	// Process
  E_SEQ_DATABASE.BUCKET_EXIST_CHECK: _m_Seq_BUCKET_EXIST_CHECK();
    IF TRUE
		AND (stSeqCtrlGeneral.eActiveSeqState = E_SEQ_GENERAL.DONE) 
		THEN
			eSeq := E_SEQ_DATABASE.BASE;
		END_IF
  
	E_SEQ_DATABASE.MEASUREMENT_EXIST_CHECK:         _m_Seq_MEASUREMENT_EXIST_CHECK();
    IF TRUE
		AND (stSeqCtrlGeneral.eActiveSeqState = E_SEQ_GENERAL.DONE) 
		THEN
			eSeq := E_SEQ_DATABASE.BASE;
		END_IF
    
  E_SEQ_DATABASE.WRITE_STRUCT:  _m_Seq_WRITE_STRUCT();
    IF TRUE
		AND (stSeqCtrlGeneral.eActiveSeqState = E_SEQ_GENERAL.DONE) 
		THEN
			eSeq := E_SEQ_DATABASE.BASE;
		END_IF
  
  E_SEQ_DATABASE.TAG_EXIST_CHECK:     _m_Seq_TAG_EXIST_CHECK();
    IF TRUE
		AND (stSeqCtrlGeneral.eActiveSeqState = E_SEQ_GENERAL.DONE) 
		THEN
			eSeq := E_SEQ_DATABASE.BASE;
		END_IF
    
  E_SEQ_DATABASE.FIELD_EXIST_CHECK:     _m_Seq_FIELD_EXIST_CHECK();
    IF TRUE
		AND (stSeqCtrlGeneral.eActiveSeqState = E_SEQ_GENERAL.DONE) 
		THEN
			eSeq := E_SEQ_DATABASE.BASE;
		END_IF
    
  E_SEQ_DATABASE.DELETE_MEASUREMENT:    _m_Seq_DELETE_MEASUREMENT();
    IF TRUE
		AND (stSeqCtrlGeneral.eActiveSeqState = E_SEQ_GENERAL.DONE) 
		THEN
			eSeq := E_SEQ_DATABASE.BASE;
		END_IF
    
  E_SEQ_DATABASE.DELETE_ALL_MEASUREMENTS:    _m_Seq_DELETE_ALL_MEASUREMENTS();
    IF TRUE
		AND (stSeqCtrlGeneral.eActiveSeqState = E_SEQ_GENERAL.DONE) 
		THEN
			eSeq := E_SEQ_DATABASE.BASE;
		END_IF
  
  E_SEQ_DATABASE.DELETE_TAG:    _m_Seq_DELETE_TAG();
    IF TRUE
		AND (stSeqCtrlGeneral.eActiveSeqState = E_SEQ_GENERAL.DONE) 
		THEN
			eSeq := E_SEQ_DATABASE.BASE;
		END_IF
    
  E_SEQ_DATABASE.DELETE_TAG_CONTENT_BLOCK:    _m_Seq_DELETE_TAG_CONTENT_BLOCK();
    IF TRUE
		AND (stSeqCtrlGeneral.eActiveSeqState = E_SEQ_GENERAL.DONE) 
		THEN
			eSeq := E_SEQ_DATABASE.BASE;
		END_IF
  
  E_SEQ_DATABASE.DELETE_FIELD:           _m_Seq_DELETE_FIELD();
    IF TRUE
		AND (stSeqCtrlGeneral.eActiveSeqState = E_SEQ_GENERAL.DONE) 
		THEN
			eSeq := E_SEQ_DATABASE.BASE;
		END_IF
    
  E_SEQ_DATABASE.GET_TOTAL_MEASUREMENTS:           _m_Seq_GET_TOTAL_MEASUREMENTS();
    IF TRUE
		AND (stSeqCtrlGeneral.eActiveSeqState = E_SEQ_GENERAL.DONE) 
		THEN
			eSeq := E_SEQ_DATABASE.BASE;
		END_IF

  // End
	E_SEQ_DATABASE.END:;
	E_SEQ_DATABASE.ERROR_SEQ:;	
END_CASE

strTemp:=TO_STRING(eSeq);

METHOD PRIVATE _m_DebugManager
VAR_INPUT
	iStepID: int;
END_VAR
IF TRUE
AND THIS^.stSeqCtrlGeneral.bDebugModeActive 
AND NOT THIS^.stSeqCtrlGeneral.bActiveStep
THEN


THIS^.stSeqCtrlGeneral.bBreakpointActive:=FALSE;

FOR i:=0 TO 10 DO
	
	IF TRUE
	AND iStepID=THIS^.stSeqCtrlGeneral.listBreakpoint[i] 
	AND iStepID<>0
	THEN
		EXIT;
	END_IF
END_FOR
IF (i<=10) THEN
	THIS^.stSeqCtrlGeneral.bBreakpointActive:=TRUE;
END_IF

END_IF
END_METHOD

METHOD PRIVATE _m_Delay : BOOL
VAR_INPUT
	DelayTime:	TIME;
END_VAR
THIS^.stSeqCtrlGeneral.bDelayActive:=TRUE;
THIS^.stSeqCtrlGeneral.tDelay:=DelayTime;
_m_Delay:=FALSE;
IF THIS^.stSeqCtrlGeneral.tonDelay.Q THEN
	_m_Delay:=TRUE;
END_IF
END_METHOD

METHOD PRIVATE _m_GeneralStepSetting : BOOL
VAR_INPUT
	StepType:			    	E_STEP_STATE_TYPE;
	InfoTextID:					STRING(20);
	EnableDebug:	   			BOOL;	
	
END_VAR
IF THIS^.stSeqCtrlGeneral.bActiveStep THEN
	THIS^.stSeqCtrlGeneral.eStep_Type:=StepType;
	THIS^.stSeqCtrlGeneral.strExtraInfo:= GenLib.F_RET_TXTLIST_ENTRY(strPortNr:='851',strID:='',strTxtLstName:=InfoTextID);
END_IF
END_METHOD

METHOD PRIVATE _m_SaveLastStep : BOOL
VAR_INPUT
END_VAR
VAR
	i: dint;
END_VAR
IF NOT THIS^.stSeqCtrlGeneral.bActiveStep THEN
	
	FOR i:=49 TO 1 BY -1 DO
			stSeqCtrlGeneral.listLastSteps[i].strStepName:=stSeqCtrlGeneral.listLastSteps[i-1].strStepName;
			stSeqCtrlGeneral.listLastSteps[i].tStepTime:=stSeqCtrlGeneral.listLastSteps[i-1].tStepTime;
			stSeqCtrlGeneral.listLastSteps[i].tDelayTime:=stSeqCtrlGeneral.listLastSteps[i-1].tDelayTime;
	END_FOR
	stSeqCtrlGeneral.listLastSteps[0].strStepName:=TO_STRING(THIS^.eSeq);
	stSeqCtrlGeneral.listLastSteps[1].tStepTime:=THIS^.stSeqCtrlGeneral.tonStepTime.ET;
	stSeqCtrlGeneral.listLastSteps[1].tStepTime:=THIS^.stSeqCtrlGeneral.tonDelay.ET;
ELSE
	stSeqCtrlGeneral.listLastSteps[0].tStepTime:=THIS^.stSeqCtrlGeneral.tonStepTime.ET;
	stSeqCtrlGeneral.listLastSteps[0].tDelayTime:=THIS^.stSeqCtrlGeneral.tonDelay.ET;	
END_IF
END_METHOD

METHOD PRIVATE _m_Seq_BUCKET_EXIST_CHECK : E_SEQ_PROCESS
VAR_INPUT
END_VAR
VAR
	ActiveSeq: STRING;
END_VAR
//THIS^._m_GeneralStepSetting(StepType:=E_STEP_STATE_TYPE.INIT,
ActiveSeq := TO_STRING(THIS^.eSeq);

CASE THIS^.stSeqCtrlGeneral.eActiveSeqState OF
E_SEQ_GENERAL.READY:;
	
E_SEQ_GENERAL.EXECUTE:;
	IF TRUE
	THEN
		THIS^.stSeqCtrlGeneral.eActiveSeqState := E_SEQ_GENERAL.RESET;
	END_IF
  
E_SEQ_GENERAL.RESET:;
	THIS^.stSeqCtrlGeneral.iInternalSeqStateCase := 0;
	IF TRUE
	THEN
    THIS^.bResult := FALSE;
		THIS^.stSeqCtrlGeneral.eActiveSeqState := E_SEQ_GENERAL.BUSY;
	END_IF
  
E_SEQ_GENERAL.BUSY:;
	CASE THIS^.stSeqCtrlGeneral.iInternalSeqStateCase OF
    0:  // Execute
      IF TRUE 
      AND THIS^.bAdsConnected
      AND NOT THIS^.bBusy
      AND THIS^.bReady
			THEN 
        THIS^.bGetBucketExist := TRUE;
        THIS^.stSeqCtrlGeneral.iInternalSeqStateCase := 10;
			END_IF

    10:	// Wait for done
      IF TRUE 
      AND NOT THIS^.bBusy
      AND THIS^.bReady
      AND NOT THIS^.bGetBucketExist
			THEN 
        THIS^.stSeqCtrlGeneral.iInternalSeqStateCase := 1000;
			END_IF
      
    1000: // Exit step
      IF TRUE
      THEN
        THIS^.stSeqCtrlGeneral.iInternalSeqStateCase := 9999;
			END_IF
      
	ELSE
		THIS^.stSeqCtrlGeneral.eActiveSeqState := E_SEQ_GENERAL.DONE;  
	END_CASE
	THIS^.stSeqCtrlGeneral.strExtraInfo := CONCAT('Internal state: ', TO_STRING(THIS^.stSeqCtrlGeneral.iInternalSeqStateCase));

E_SEQ_GENERAL.DONE:;

E_SEQ_GENERAL.ERROR:;

E_SEQ_GENERAL.TIME_OUT:; 

ELSE
  THIS^.stSeqCtrlGeneral.eActiveSeqState := E_SEQ_GENERAL.ERROR;
END_CASE
END_METHOD

METHOD PRIVATE _m_Seq_CLEAR_MEASUREMENT : E_SEQ_PROCESS
VAR_INPUT
END_VAR
VAR
	ActiveSeq: STRING;
END_VAR
//THIS^._m_GeneralStepSetting(StepType:=E_STEP_STATE_TYPE.INIT,
ActiveSeq := TO_STRING(THIS^.eSeq);

CASE THIS^.stSeqCtrlGeneral.eActiveSeqState OF
E_SEQ_GENERAL.READY:;
	
E_SEQ_GENERAL.EXECUTE:;
	IF TRUE
	THEN
		THIS^.stSeqCtrlGeneral.eActiveSeqState := E_SEQ_GENERAL.RESET;
	END_IF
  
E_SEQ_GENERAL.RESET:;
	THIS^.stSeqCtrlGeneral.iInternalSeqStateCase := 0;
	IF TRUE
	THEN
    THIS^.bResult := FALSE;
		THIS^.stSeqCtrlGeneral.eActiveSeqState := E_SEQ_GENERAL.BUSY;
	END_IF
  
E_SEQ_GENERAL.BUSY:;
	CASE THIS^.stSeqCtrlGeneral.iInternalSeqStateCase OF
		0:	// Entrance step --> Create command
      IF TRUE 
      AND THIS^.bAdsConnected
      AND NOT THIS^.bBusy
      AND THIS^.bReady
			THEN 
        THIS^.bClearMeasurement := TRUE;
        THIS^.stSeqCtrlGeneral.iInternalSeqStateCase := 10;
			END_IF
      
    10:	// Wait for done
      IF TRUE 
      AND NOT THIS^.bBusy
      AND THIS^.bReady
      AND NOT THIS^.bClearMeasurement
			THEN 
        THIS^.stSeqCtrlGeneral.iInternalSeqStateCase := 1000;
			END_IF
      
    1000: // Exit step
      IF TRUE
      THEN
        THIS^.stSeqCtrlGeneral.iInternalSeqStateCase := 9999;
			END_IF
      
	ELSE
		THIS^.stSeqCtrlGeneral.eActiveSeqState := E_SEQ_GENERAL.DONE;  
	END_CASE
	THIS^.stSeqCtrlGeneral.strExtraInfo := CONCAT('Internal state: ', TO_STRING(THIS^.stSeqCtrlGeneral.iInternalSeqStateCase));

E_SEQ_GENERAL.DONE:;

E_SEQ_GENERAL.ERROR:;

E_SEQ_GENERAL.TIME_OUT:; 
IF TRUE
AND THIS^.stSeqCtrlGeneral.bTimeOutActiveQuit 
THEN
  THIS^.stSeqCtrlGeneral.strExtraInfo := 'Bitte quittieren und erneut testen';
  IF TRUE
  //AND itfOpMode.P_QUIT
  THEN
    THIS^.stSeqCtrlGeneral.eActiveSeqState := E_SEQ_GENERAL.EXECUTE;
	END_IF
  
END_IF

ELSE
  THIS^.stSeqCtrlGeneral.eActiveSeqState := E_SEQ_GENERAL.ERROR;
END_CASE
END_METHOD

METHOD PRIVATE _m_Seq_DELETE_ALL_MEASUREMENTS : E_SEQ_PROCESS
VAR_INPUT
END_VAR
VAR
	ActiveSeq: STRING;
END_VAR
//THIS^._m_GeneralStepSetting(StepType:=E_STEP_STATE_TYPE.INIT,
ActiveSeq := TO_STRING(THIS^.eSeq);

CASE THIS^.stSeqCtrlGeneral.eActiveSeqState OF
E_SEQ_GENERAL.READY:;

E_SEQ_GENERAL.EXECUTE:;
	IF TRUE
	THEN
		THIS^.stSeqCtrlGeneral.eActiveSeqState := E_SEQ_GENERAL.RESET;
	END_IF
  
E_SEQ_GENERAL.RESET:;
	THIS^.stSeqCtrlGeneral.iInternalSeqStateCase := 0;
	IF TRUE
	THEN
    THIS^.bResult := FALSE;
		THIS^.stSeqCtrlGeneral.eActiveSeqState := E_SEQ_GENERAL.BUSY;
	END_IF
  
E_SEQ_GENERAL.BUSY:;
	CASE THIS^.stSeqCtrlGeneral.iInternalSeqStateCase OF
		0:	// Entrance step --> Create command
      IF TRUE 
      AND THIS^.bAdsConnected
      AND NOT THIS^.bBusy
      AND THIS^.bReady
			THEN 
        THIS^.bDeleteAllMeasurements := TRUE;
        THIS^.stSeqCtrlGeneral.iInternalSeqStateCase := 10;
			END_IF
      
    10:	// Wait for done
      IF TRUE 
      AND NOT THIS^.bBusy
      AND THIS^.bReady
      AND NOT THIS^.bDeleteAllMeasurements
			THEN 
        THIS^.stSeqCtrlGeneral.iInternalSeqStateCase := 1000;
			END_IF
      
    1000: // Exit step
      IF TRUE
      THEN
        THIS^.stSeqCtrlGeneral.iInternalSeqStateCase := 9999;
			END_IF
      
	ELSE
		THIS^.stSeqCtrlGeneral.eActiveSeqState := E_SEQ_GENERAL.DONE;  
	END_CASE
	THIS^.stSeqCtrlGeneral.strExtraInfo := CONCAT('Internal state: ', TO_STRING(THIS^.stSeqCtrlGeneral.iInternalSeqStateCase));

E_SEQ_GENERAL.DONE:;

E_SEQ_GENERAL.ERROR:;

E_SEQ_GENERAL.TIME_OUT:; 
IF TRUE
AND THIS^.stSeqCtrlGeneral.bTimeOutActiveQuit 
THEN
  THIS^.stSeqCtrlGeneral.strExtraInfo := 'Bitte quittieren und erneut testen';
  IF TRUE
  //AND itfOpMode.P_QUIT
  THEN
    THIS^.stSeqCtrlGeneral.eActiveSeqState := E_SEQ_GENERAL.EXECUTE;
	END_IF
  
END_IF

ELSE
  THIS^.stSeqCtrlGeneral.eActiveSeqState := E_SEQ_GENERAL.ERROR;
END_CASE
END_METHOD

METHOD PRIVATE _m_Seq_DELETE_FIELD : E_SEQ_PROCESS
VAR_INPUT
END_VAR
VAR
	ActiveSeq: STRING;
END_VAR
//THIS^._m_GeneralStepSetting(StepType:=E_STEP_STATE_TYPE.INIT,
ActiveSeq := TO_STRING(THIS^.eSeq);

CASE THIS^.stSeqCtrlGeneral.eActiveSeqState OF
E_SEQ_GENERAL.READY:;
	
E_SEQ_GENERAL.EXECUTE:;
	IF TRUE
	THEN
		THIS^.stSeqCtrlGeneral.eActiveSeqState := E_SEQ_GENERAL.RESET;
	END_IF
  
E_SEQ_GENERAL.RESET:;
	THIS^.stSeqCtrlGeneral.iInternalSeqStateCase := 0;
	IF TRUE
	THEN
    THIS^.bResult := FALSE;
		THIS^.stSeqCtrlGeneral.eActiveSeqState := E_SEQ_GENERAL.BUSY;
	END_IF
  
E_SEQ_GENERAL.BUSY:;
	CASE THIS^.stSeqCtrlGeneral.iInternalSeqStateCase OF
    0:  // Execute
      IF TRUE 
      AND THIS^.bAdsConnected
      AND NOT THIS^.bBusy
      AND THIS^.bReady
			THEN 
        THIS^.bDeleteField := TRUE;
        THIS^.stSeqCtrlGeneral.iInternalSeqStateCase := 10;
			END_IF

    10:	// Wait for done
      IF TRUE 
      AND NOT THIS^.bBusy
      AND THIS^.bReady
      AND NOT THIS^.bDeleteField
			THEN 
        THIS^.stSeqCtrlGeneral.iInternalSeqStateCase := 1000;
			END_IF
      
    1000: // Exit step
      IF TRUE
      THEN
        THIS^.stSeqCtrlGeneral.iInternalSeqStateCase := 9999;
			END_IF
      
	ELSE
		THIS^.stSeqCtrlGeneral.eActiveSeqState := E_SEQ_GENERAL.DONE;  
	END_CASE
	THIS^.stSeqCtrlGeneral.strExtraInfo := CONCAT('Internal state: ', TO_STRING(THIS^.stSeqCtrlGeneral.iInternalSeqStateCase));

E_SEQ_GENERAL.DONE:;

E_SEQ_GENERAL.ERROR:;

E_SEQ_GENERAL.TIME_OUT:; 

ELSE
  THIS^.stSeqCtrlGeneral.eActiveSeqState := E_SEQ_GENERAL.ERROR;
END_CASE
END_METHOD

METHOD PRIVATE _m_Seq_DELETE_MEASUREMENT : E_SEQ_PROCESS
VAR_INPUT
END_VAR
VAR
	ActiveSeq: STRING;
END_VAR
//THIS^._m_GeneralStepSetting(StepType:=E_STEP_STATE_TYPE.INIT,
ActiveSeq := TO_STRING(THIS^.eSeq);

CASE THIS^.stSeqCtrlGeneral.eActiveSeqState OF
E_SEQ_GENERAL.READY:;
	
E_SEQ_GENERAL.EXECUTE:;
	IF TRUE
	THEN
		THIS^.stSeqCtrlGeneral.eActiveSeqState := E_SEQ_GENERAL.RESET;
	END_IF
  
E_SEQ_GENERAL.RESET:;
	THIS^.stSeqCtrlGeneral.iInternalSeqStateCase := 0;
	IF TRUE
	THEN
    THIS^.bResult := FALSE;
		THIS^.stSeqCtrlGeneral.eActiveSeqState := E_SEQ_GENERAL.BUSY;
	END_IF
  
E_SEQ_GENERAL.BUSY:;
	CASE THIS^.stSeqCtrlGeneral.iInternalSeqStateCase OF
		0:	// Entrance step --> Create command
      IF TRUE 
      AND THIS^.bAdsConnected
      AND NOT THIS^.bBusy
      AND THIS^.bReady
			THEN 
        THIS^.bDeleteMeasurement := TRUE;
        THIS^.stSeqCtrlGeneral.iInternalSeqStateCase := 10;
			END_IF
      
    10:	// Wait for done
      IF TRUE 
      AND NOT THIS^.bBusy
      AND THIS^.bReady
      AND NOT THIS^.bDeleteMeasurement
			THEN 
        THIS^.stSeqCtrlGeneral.iInternalSeqStateCase := 1000;
			END_IF
      
    1000: // Exit step
      IF TRUE
      THEN
        THIS^.stSeqCtrlGeneral.iInternalSeqStateCase := 9999;
			END_IF
      
	ELSE
		THIS^.stSeqCtrlGeneral.eActiveSeqState := E_SEQ_GENERAL.DONE;  
	END_CASE
	THIS^.stSeqCtrlGeneral.strExtraInfo := CONCAT('Internal state: ', TO_STRING(THIS^.stSeqCtrlGeneral.iInternalSeqStateCase));

E_SEQ_GENERAL.DONE:;

E_SEQ_GENERAL.ERROR:;

E_SEQ_GENERAL.TIME_OUT:; 
IF TRUE
AND THIS^.stSeqCtrlGeneral.bTimeOutActiveQuit 
THEN
  THIS^.stSeqCtrlGeneral.strExtraInfo := 'Bitte quittieren und erneut testen';
  IF TRUE
  //AND itfOpMode.P_QUIT
  THEN
    THIS^.stSeqCtrlGeneral.eActiveSeqState := E_SEQ_GENERAL.EXECUTE;
	END_IF
  
END_IF

ELSE
  THIS^.stSeqCtrlGeneral.eActiveSeqState := E_SEQ_GENERAL.ERROR;
END_CASE
END_METHOD

METHOD PRIVATE _m_Seq_DELETE_TAG : E_SEQ_PROCESS
VAR_INPUT
END_VAR
VAR
	ActiveSeq: STRING;
END_VAR
//THIS^._m_GeneralStepSetting(StepType:=E_STEP_STATE_TYPE.INIT,
ActiveSeq := TO_STRING(THIS^.eSeq);

CASE THIS^.stSeqCtrlGeneral.eActiveSeqState OF
E_SEQ_GENERAL.READY:;
	
E_SEQ_GENERAL.EXECUTE:;
	IF TRUE
	THEN
		THIS^.stSeqCtrlGeneral.eActiveSeqState := E_SEQ_GENERAL.RESET;
	END_IF
  
E_SEQ_GENERAL.RESET:;
	THIS^.stSeqCtrlGeneral.iInternalSeqStateCase := 0;
	IF TRUE
	THEN
    THIS^.bResult := FALSE;
		THIS^.stSeqCtrlGeneral.eActiveSeqState := E_SEQ_GENERAL.BUSY;
	END_IF
  
E_SEQ_GENERAL.BUSY:;
	CASE THIS^.stSeqCtrlGeneral.iInternalSeqStateCase OF
    0:  // Execute
      IF TRUE 
      AND THIS^.bAdsConnected
      AND NOT THIS^.bBusy
      AND THIS^.bReady
			THEN 
        THIS^.bDeleteTag := TRUE;
        THIS^.stSeqCtrlGeneral.iInternalSeqStateCase := 10;
			END_IF

    10:	// Wait for done
      IF TRUE 
      AND NOT THIS^.bBusy
      AND THIS^.bReady
      AND NOT THIS^.bDeleteTag
			THEN 
        THIS^.stSeqCtrlGeneral.iInternalSeqStateCase := 1000;
			END_IF
      
    1000: // Exit step
      IF TRUE
      THEN
        THIS^.stSeqCtrlGeneral.iInternalSeqStateCase := 9999;
			END_IF
      
	ELSE
		THIS^.stSeqCtrlGeneral.eActiveSeqState := E_SEQ_GENERAL.DONE;  
	END_CASE
	THIS^.stSeqCtrlGeneral.strExtraInfo := CONCAT('Internal state: ', TO_STRING(THIS^.stSeqCtrlGeneral.iInternalSeqStateCase));

E_SEQ_GENERAL.DONE:;

E_SEQ_GENERAL.ERROR:;

E_SEQ_GENERAL.TIME_OUT:; 

ELSE
  THIS^.stSeqCtrlGeneral.eActiveSeqState := E_SEQ_GENERAL.ERROR;
END_CASE
END_METHOD

METHOD PRIVATE _m_Seq_DELETE_TAG_CONTENT_BLOCK : E_SEQ_PROCESS
VAR_INPUT
END_VAR
VAR
	ActiveSeq: STRING;
END_VAR
//THIS^._m_GeneralStepSetting(StepType:=E_STEP_STATE_TYPE.INIT,
ActiveSeq := TO_STRING(THIS^.eSeq);

CASE THIS^.stSeqCtrlGeneral.eActiveSeqState OF
E_SEQ_GENERAL.READY:;
	
E_SEQ_GENERAL.EXECUTE:;
	IF TRUE
	THEN
		THIS^.stSeqCtrlGeneral.eActiveSeqState := E_SEQ_GENERAL.RESET;
	END_IF
  
E_SEQ_GENERAL.RESET:;
	THIS^.stSeqCtrlGeneral.iInternalSeqStateCase := 0;
	IF TRUE
	THEN
    THIS^.bResult := FALSE;
		THIS^.stSeqCtrlGeneral.eActiveSeqState := E_SEQ_GENERAL.BUSY;
	END_IF
  
E_SEQ_GENERAL.BUSY:;
	CASE THIS^.stSeqCtrlGeneral.iInternalSeqStateCase OF
    0:  // Execute
      IF TRUE 
      AND THIS^.bAdsConnected
      AND NOT THIS^.bBusy
      AND THIS^.bReady
			THEN 
        THIS^.bDeleteTagContentBlock := TRUE;
        THIS^.stSeqCtrlGeneral.iInternalSeqStateCase := 10;
			END_IF

    10:	// Wait for done
      IF TRUE 
      AND NOT THIS^.bBusy
      AND THIS^.bReady
      AND NOT THIS^.bDeleteTagContentBlock
			THEN 
        THIS^.stSeqCtrlGeneral.iInternalSeqStateCase := 1000;
			END_IF
      
    1000: // Exit step
      IF TRUE
      THEN
        THIS^.stSeqCtrlGeneral.iInternalSeqStateCase := 9999;
			END_IF
      
	ELSE
		THIS^.stSeqCtrlGeneral.eActiveSeqState := E_SEQ_GENERAL.DONE;  
	END_CASE
	THIS^.stSeqCtrlGeneral.strExtraInfo := CONCAT('Internal state: ', TO_STRING(THIS^.stSeqCtrlGeneral.iInternalSeqStateCase));

E_SEQ_GENERAL.DONE:;

E_SEQ_GENERAL.ERROR:;

E_SEQ_GENERAL.TIME_OUT:; 

ELSE
  THIS^.stSeqCtrlGeneral.eActiveSeqState := E_SEQ_GENERAL.ERROR;
END_CASE
END_METHOD

METHOD PRIVATE _m_Seq_FIELD_EXIST_CHECK : E_SEQ_PROCESS
VAR_INPUT
END_VAR
VAR
	ActiveSeq: STRING;
END_VAR
//THIS^._m_GeneralStepSetting(StepType:=E_STEP_STATE_TYPE.INIT,
ActiveSeq := TO_STRING(THIS^.eSeq);

CASE THIS^.stSeqCtrlGeneral.eActiveSeqState OF
E_SEQ_GENERAL.READY:;
	
E_SEQ_GENERAL.EXECUTE:;
	IF TRUE
	THEN
		THIS^.stSeqCtrlGeneral.eActiveSeqState := E_SEQ_GENERAL.RESET;
	END_IF
  
E_SEQ_GENERAL.RESET:;
	THIS^.stSeqCtrlGeneral.iInternalSeqStateCase := 0;
	IF TRUE
	THEN
    THIS^.bResult := FALSE;
		THIS^.stSeqCtrlGeneral.eActiveSeqState := E_SEQ_GENERAL.BUSY;
	END_IF
  
E_SEQ_GENERAL.BUSY:;
	CASE THIS^.stSeqCtrlGeneral.iInternalSeqStateCase OF
    0:  // Execute
      IF TRUE 
      AND THIS^.bAdsConnected
      AND NOT THIS^.bBusy
      AND THIS^.bReady
			THEN 
        THIS^.bGetFieldExist := TRUE;
        THIS^.stSeqCtrlGeneral.iInternalSeqStateCase := 10;
			END_IF

    10:	// Wait for done
      IF TRUE 
      AND NOT THIS^.bBusy
      AND THIS^.bReady
      AND NOT THIS^.bGetFieldExist
			THEN 
        THIS^.stSeqCtrlGeneral.iInternalSeqStateCase := 1000;
			END_IF
      
    1000: // Exit step
      IF TRUE
      THEN
        THIS^.stSeqCtrlGeneral.iInternalSeqStateCase := 9999;
			END_IF
      
	ELSE
		THIS^.stSeqCtrlGeneral.eActiveSeqState := E_SEQ_GENERAL.DONE;  
	END_CASE
	THIS^.stSeqCtrlGeneral.strExtraInfo := CONCAT('Internal state: ', TO_STRING(THIS^.stSeqCtrlGeneral.iInternalSeqStateCase));

E_SEQ_GENERAL.DONE:;

E_SEQ_GENERAL.ERROR:;

E_SEQ_GENERAL.TIME_OUT:; 

ELSE
  THIS^.stSeqCtrlGeneral.eActiveSeqState := E_SEQ_GENERAL.ERROR;
END_CASE
END_METHOD

METHOD PRIVATE _m_Seq_GET_TOTAL_MEASUREMENTS : E_SEQ_PROCESS
VAR_INPUT
END_VAR
VAR
	ActiveSeq: STRING;
END_VAR
//THIS^._m_GeneralStepSetting(StepType:=E_STEP_STATE_TYPE.INIT,
ActiveSeq := TO_STRING(THIS^.eSeq);

CASE THIS^.stSeqCtrlGeneral.eActiveSeqState OF
E_SEQ_GENERAL.READY:;
	
E_SEQ_GENERAL.EXECUTE:;
	IF TRUE
	THEN
		THIS^.stSeqCtrlGeneral.eActiveSeqState := E_SEQ_GENERAL.RESET;
	END_IF
  
E_SEQ_GENERAL.RESET:;
	THIS^.stSeqCtrlGeneral.iInternalSeqStateCase := 0;
	IF TRUE
	THEN
    THIS^.bResult := FALSE;
		THIS^.stSeqCtrlGeneral.eActiveSeqState := E_SEQ_GENERAL.BUSY;
	END_IF
  
E_SEQ_GENERAL.BUSY:;
	CASE THIS^.stSeqCtrlGeneral.iInternalSeqStateCase OF
    0:  // Execute
      IF TRUE 
      AND THIS^.bAdsConnected
      AND NOT THIS^.bBusy
      AND THIS^.bReady
			THEN 
        THIS^.bGetTotalMeasurements := TRUE;
        THIS^.stSeqCtrlGeneral.iInternalSeqStateCase := 10;
			END_IF

    10:	// Wait for done
      IF TRUE 
      AND NOT THIS^.bBusy
      AND THIS^.bReady
      AND NOT THIS^.bGetTotalMeasurements
			THEN 
        THIS^.stSeqCtrlGeneral.iInternalSeqStateCase := 1000;
			END_IF
      
    1000: // Exit step
      IF TRUE
      THEN
        THIS^.stSeqCtrlGeneral.iInternalSeqStateCase := 9999;
			END_IF
      
	ELSE
		THIS^.stSeqCtrlGeneral.eActiveSeqState := E_SEQ_GENERAL.DONE;  
	END_CASE
	THIS^.stSeqCtrlGeneral.strExtraInfo := CONCAT('Internal state: ', TO_STRING(THIS^.stSeqCtrlGeneral.iInternalSeqStateCase));

E_SEQ_GENERAL.DONE:;

E_SEQ_GENERAL.ERROR:;

E_SEQ_GENERAL.TIME_OUT:; 

ELSE
  THIS^.stSeqCtrlGeneral.eActiveSeqState := E_SEQ_GENERAL.ERROR;
END_CASE
END_METHOD

METHOD PRIVATE _m_Seq_INIT : E_SEQ_PROCESS
VAR_INPUT
END_VAR
VAR
	ActiveSeq: STRING;
END_VAR
VAR
	
END_VAR
//THIS^._m_GeneralStepSetting(StepType:=E_STEP_STATE_TYPE.INIT,
ActiveSeq := TO_STRING(THIS^.eSeq);

CASE THIS^.stSeqCtrlGeneral.eActiveSeqState OF
E_SEQ_GENERAL.READY:;
	
E_SEQ_GENERAL.EXECUTE:;
	IF TRUE
	THEN
		THIS^.stSeqCtrlGeneral.eActiveSeqState := E_SEQ_GENERAL.RESET;
	END_IF
E_SEQ_GENERAL.RESET:;
	THIS^.stSeqCtrlGeneral.iInternalSeqStateCase := 0;
	IF TRUE
	THEN
		THIS^.stSeqCtrlGeneral.eActiveSeqState := E_SEQ_GENERAL.BUSY;
	END_IF
E_SEQ_GENERAL.BUSY:;
	CASE THIS^.stSeqCtrlGeneral.iInternalSeqStateCase OF
		0:	// Entrance step
      IF TRUE
			THEN 
        THIS^.bResult := FALSE;
        THIS^.bGetBucketExist := FALSE;
        THIS^.sBucketName := '';
        THIS^.bGetMeasurementExist := FALSE;
        THIS^.sMeasurementName := '';
        THIS^.bDeleteMeasurement := FALSE;
        THIS^.bDeleteAllMeasurements := FALSE;
        THIS^.bWriteStructData := FALSE;
        THIS^.sTagName := '';
        THIS^.sFieldName := '';
        //THIS^.stFieldValues := '';
        //FOR THIS^.i := 0 TO TO_INT(SIZEOF(arrFieldNames)) BY 1 DO
        //  THIS^.arrFieldNames[i] := '';
        //  THIS^.arrFieldStructContent[i] := '';
        //END_FOR
        THIS^.dtFrom := DT#1970-1-1-0:0:0;
        THIS^.dtTo := DT#1970-1-1-0:0:0;
				THIS^.stSeqCtrlGeneral.iInternalSeqStateCase := 1000;
			END_IF
      
    1000:	// Exit step
      IF TRUE
			THEN
        THIS^.stSeqCtrlGeneral.iInternalSeqStateCase := 9999;
      END_IF
      
	ELSE
		THIS^.stSeqCtrlGeneral.eActiveSeqState := E_SEQ_GENERAL.DONE;  
	END_CASE
	THIS^.stSeqCtrlGeneral.strExtraInfo := CONCAT('Internal state: ', TO_STRING(THIS^.stSeqCtrlGeneral.iInternalSeqStateCase));
E_SEQ_GENERAL.DONE:;
E_SEQ_GENERAL.ERROR:;
E_SEQ_GENERAL.TIME_OUT:; 

IF TRUE
AND THIS^.stSeqCtrlGeneral.bTimeOutActiveQuit 
THEN
  THIS^.stSeqCtrlGeneral.strExtraInfo := 'Bitte quittieren und erneut testen';
  IF TRUE
  //AND itfOpMode.P_QUIT
  THEN
    THIS^.stSeqCtrlGeneral.eActiveSeqState := E_SEQ_GENERAL.EXECUTE;
	END_IF
  
END_IF

ELSE
  THIS^.stSeqCtrlGeneral.eActiveSeqState := E_SEQ_GENERAL.ERROR;
END_CASE
END_METHOD

METHOD PRIVATE _m_Seq_MEASUREMENT_EXIST_CHECK : E_SEQ_PROCESS
VAR_INPUT
END_VAR
VAR
	ActiveSeq: STRING;
END_VAR
//THIS^._m_GeneralStepSetting(StepType:=E_STEP_STATE_TYPE.INIT,
ActiveSeq := TO_STRING(THIS^.eSeq);

CASE THIS^.stSeqCtrlGeneral.eActiveSeqState OF
E_SEQ_GENERAL.READY:;
	
E_SEQ_GENERAL.EXECUTE:;
	IF TRUE
	THEN
		THIS^.stSeqCtrlGeneral.eActiveSeqState := E_SEQ_GENERAL.RESET;
	END_IF
  
E_SEQ_GENERAL.RESET:;
	THIS^.stSeqCtrlGeneral.iInternalSeqStateCase := 0;
	IF TRUE
	THEN
    THIS^.bResult := FALSE;
		THIS^.stSeqCtrlGeneral.eActiveSeqState := E_SEQ_GENERAL.BUSY;
	END_IF
  
E_SEQ_GENERAL.BUSY:;
	CASE THIS^.stSeqCtrlGeneral.iInternalSeqStateCase OF
    0:  // Execute
      IF TRUE 
      AND THIS^.bAdsConnected
      AND NOT THIS^.bBusy
      AND THIS^.bReady
			THEN 
        THIS^.bGetMeasurementExist := TRUE;
        THIS^.stSeqCtrlGeneral.iInternalSeqStateCase := 10;
			END_IF

    10:	// Wait for done
      IF TRUE 
      AND NOT THIS^.bBusy
      AND THIS^.bReady
      AND NOT THIS^.bGetMeasurementExist
			THEN 
        THIS^.stSeqCtrlGeneral.iInternalSeqStateCase := 1000;
			END_IF
      
    1000: // Exit step
      IF TRUE
      THEN
        THIS^.stSeqCtrlGeneral.iInternalSeqStateCase := 9999;
			END_IF
      
	ELSE
		THIS^.stSeqCtrlGeneral.eActiveSeqState := E_SEQ_GENERAL.DONE;  
	END_CASE
	THIS^.stSeqCtrlGeneral.strExtraInfo := CONCAT('Internal state: ', TO_STRING(THIS^.stSeqCtrlGeneral.iInternalSeqStateCase));

E_SEQ_GENERAL.DONE:;

E_SEQ_GENERAL.ERROR:;

E_SEQ_GENERAL.TIME_OUT:; 

ELSE
  THIS^.stSeqCtrlGeneral.eActiveSeqState := E_SEQ_GENERAL.ERROR;
END_CASE
END_METHOD

METHOD PRIVATE _m_Seq_TAG_EXIST_CHECK : E_SEQ_PROCESS
VAR_INPUT
END_VAR
VAR
	ActiveSeq: STRING;
END_VAR
//THIS^._m_GeneralStepSetting(StepType:=E_STEP_STATE_TYPE.INIT,
ActiveSeq := TO_STRING(THIS^.eSeq);

CASE THIS^.stSeqCtrlGeneral.eActiveSeqState OF
E_SEQ_GENERAL.READY:;
	
E_SEQ_GENERAL.EXECUTE:;
	IF TRUE
	THEN
		THIS^.stSeqCtrlGeneral.eActiveSeqState := E_SEQ_GENERAL.RESET;
	END_IF
  
E_SEQ_GENERAL.RESET:;
	THIS^.stSeqCtrlGeneral.iInternalSeqStateCase := 0;
	IF TRUE
	THEN
    THIS^.bResult := FALSE;
		THIS^.stSeqCtrlGeneral.eActiveSeqState := E_SEQ_GENERAL.BUSY;
	END_IF
  
E_SEQ_GENERAL.BUSY:;
	CASE THIS^.stSeqCtrlGeneral.iInternalSeqStateCase OF
    0:  // Execute
      IF TRUE 
      AND THIS^.bAdsConnected
      AND NOT THIS^.bBusy
      AND THIS^.bReady
			THEN 
        THIS^.bGetTagExist := TRUE;
        THIS^.stSeqCtrlGeneral.iInternalSeqStateCase := 10;
			END_IF

    10:	// Wait for done
      IF TRUE 
      AND NOT THIS^.bBusy
      AND THIS^.bReady
      AND NOT THIS^.bGetTagExist
			THEN 
        THIS^.stSeqCtrlGeneral.iInternalSeqStateCase := 1000;
			END_IF
      
    1000: // Exit step
      IF TRUE
      THEN
        THIS^.stSeqCtrlGeneral.iInternalSeqStateCase := 9999;
			END_IF
      
	ELSE
		THIS^.stSeqCtrlGeneral.eActiveSeqState := E_SEQ_GENERAL.DONE;  
	END_CASE
	THIS^.stSeqCtrlGeneral.strExtraInfo := CONCAT('Internal state: ', TO_STRING(THIS^.stSeqCtrlGeneral.iInternalSeqStateCase));

E_SEQ_GENERAL.DONE:;

E_SEQ_GENERAL.ERROR:;

E_SEQ_GENERAL.TIME_OUT:; 

ELSE
  THIS^.stSeqCtrlGeneral.eActiveSeqState := E_SEQ_GENERAL.ERROR;
END_CASE
END_METHOD

METHOD PRIVATE _m_Seq_WRITE_STRUCT : E_SEQ_PROCESS
VAR_INPUT
END_VAR
VAR
	ActiveSeq: STRING;
END_VAR
//THIS^._m_GeneralStepSetting(StepType:=E_STEP_STATE_TYPE.INIT,
ActiveSeq := TO_STRING(THIS^.eSeq);

CASE THIS^.stSeqCtrlGeneral.eActiveSeqState OF
E_SEQ_GENERAL.READY:;

	
E_SEQ_GENERAL.EXECUTE:;
	IF TRUE
	THEN
		THIS^.stSeqCtrlGeneral.eActiveSeqState := E_SEQ_GENERAL.RESET;
	END_IF
  
E_SEQ_GENERAL.RESET:;
	THIS^.stSeqCtrlGeneral.iInternalSeqStateCase := 0;
	IF TRUE
	THEN
    THIS^.bResult := FALSE;
		THIS^.stSeqCtrlGeneral.eActiveSeqState := E_SEQ_GENERAL.BUSY;
	END_IF
  
E_SEQ_GENERAL.BUSY:;
	CASE THIS^.stSeqCtrlGeneral.iInternalSeqStateCase OF
		0:	// Entrance step --> Create command
      IF TRUE 
      AND THIS^.bAdsConnected
      AND NOT THIS^.bBusy
      AND THIS^.bReady
			THEN 
        THIS^.bWriteStructData := TRUE;
        THIS^.stSeqCtrlGeneral.iInternalSeqStateCase := 10;
			END_IF
      
    10:	// Wait for done
      IF TRUE 
      AND NOT THIS^.bBusy
      AND THIS^.bReady
      AND NOT THIS^.bWriteStructData
			THEN 
        THIS^.stSeqCtrlGeneral.iInternalSeqStateCase := 1000;
			END_IF
      
    1000: // Exit step
      IF TRUE
      THEN
        THIS^.stSeqCtrlGeneral.iInternalSeqStateCase := 9999;
			END_IF
      
	ELSE
		THIS^.stSeqCtrlGeneral.eActiveSeqState := E_SEQ_GENERAL.DONE;  
	END_CASE
	THIS^.stSeqCtrlGeneral.strExtraInfo := CONCAT('Internal state: ', TO_STRING(THIS^.stSeqCtrlGeneral.iInternalSeqStateCase));

E_SEQ_GENERAL.DONE:;

E_SEQ_GENERAL.ERROR:;

E_SEQ_GENERAL.TIME_OUT:; 
IF TRUE
AND THIS^.stSeqCtrlGeneral.bTimeOutActiveQuit 
THEN
  THIS^.stSeqCtrlGeneral.strExtraInfo := 'Bitte quittieren und erneut testen';
  IF TRUE
  //AND itfOpMode.P_QUIT
  THEN
    THIS^.stSeqCtrlGeneral.eActiveSeqState := E_SEQ_GENERAL.EXECUTE;
	END_IF
  
END_IF

ELSE
  THIS^.stSeqCtrlGeneral.eActiveSeqState := E_SEQ_GENERAL.ERROR;
END_CASE
END_METHOD

METHOD PRIVATE _m_SequenceManager
VAR_INPUT
END_VAR
IF FALSE
//AND THIS^.eActiveSeqState=DONE 
AND eLastSeq<>eSeq
THEN
	IF THIS^.stSeqCtrlGeneral.eActiveSeqState<>E_SEQ_GENERAL.EXECUTE THEN
		THIS^.stSeqCtrlGeneral.eActiveSeqState:=E_SEQ_GENERAL.READY;
	END_IF
END_IF

eSeq := eNextSeq;

//DelayTimer und TimeOut Timer verwalten
stSeqCtrlGeneral.bActiveStep:=	TRUE
				AND eLastSeq					=	eSeq
				AND stSeqCtrlGeneral.eLastActiveSeqState			=	stSeqCtrlGeneral.eActiveSeqState
				AND	stSeqCtrlGeneral.iLastInternalSeqStateCase	=	stSeqCtrlGeneral.iInternalSeqStateCase
				;
			
IF NOT stSeqCtrlGeneral.bActiveStep THEN
	stSeqCtrlGeneral.bDelayActive:=FALSE;
	stSeqCtrlGeneral.bTimeOutActiveQuit:=FALSE;
	stSeqCtrlGeneral.bTimeOutActiveNoQuit:=FALSE;
  THIS^.stSeqCtrlGeneral.strExtraInfo:='';
END_IF

_m_SaveLastStep();
stSeqCtrlGeneral.tonDelay	(IN:=stSeqCtrlGeneral.bActiveStep AND stSeqCtrlGeneral.bDelayActive, 		PT:=stSeqCtrlGeneral.tDelay);
stSeqCtrlGeneral.tonTimeOut	(IN:=stSeqCtrlGeneral.bActiveStep AND (stSeqCtrlGeneral.bTimeOutActiveNoQuit OR stSeqCtrlGeneral.bTimeOutActiveQuit), 	PT:=stSeqCtrlGeneral.tTimeOut);
stSeqCtrlGeneral.tonStepTime	(IN:= stSeqCtrlGeneral.bActiveStep, PT:= T#24H);

IF stSeqCtrlGeneral.tonTimeOut.Q  THEN
	stSeqCtrlGeneral.eActiveSeqState:=E_SEQ_GENERAL.TIME_OUT;
END_IF

IF stSeqCtrlGeneral.iError<>0 THEN
	eSeq:=E_SEQ_DATABASE.ERROR_SEQ;
END_IF



eLastSeq					:=	eSeq;
stSeqCtrlGeneral.eLastActiveSeqState			:=	stSeqCtrlGeneral.eActiveSeqState;
stSeqCtrlGeneral.iLastInternalSeqStateCase	:=	stSeqCtrlGeneral.iInternalSeqStateCase;

// Reset set ready state
IF THIS^.stSeqCtrlGeneral.bExitSetReadyState THEN
  THIS^.stSeqCtrlGeneral.bExitSetReadyState := FALSE;
END_IF
END_METHOD

METHOD PRIVATE _m_TimeOut : BOOL
VAR_INPUT
	bTimeoutActiveToQuit:	BOOL;
	bTimeOutActiveNoQuit:	BOOL;
	tTimeOut:				TIME;	
END_VAR
THIS^.stSeqCtrlGeneral.bTimeOutActiveQuit:=	bTimeoutActiveToQuit;
THIS^.stSeqCtrlGeneral.bTimeOutActiveNoQuit:=	bTimeOutActiveNoQuit;
THIS^.stSeqCtrlGeneral.tTimeOut:=			tTimeOut;
_m_TimeOut:=FALSE;
IF THIS^.stSeqCtrlGeneral.tonTimeOut.Q THEN
	_m_TimeOut:=TRUE;
END_IF
END_METHOD

ACTION A_010_ADSState:
tonADSState(IN:= NOT bResetADSStateTimer, PT:= tLifeBitTimeout);
bResetADSStateTimer := FALSE;
tonADSState.IN := TRUE;

CASE uiADSStateSeq OF
  0:
    IF bADSLifeBit AND bAdsConnected THEN
      bResetADSStateTimer := TRUE;
      bADSState := TRUE;
      uiADSStateSeq := 1;
    ELSIF tonADSState.Q THEN
      stSeqCtrlGeneral.eActiveSeqState := E_SEQ_GENERAL.ERROR;
      bADSState := FALSE;
		END_IF
  1:
    IF NOT bADSLifeBit AND bAdsConnected THEN
      bResetADSStateTimer := TRUE;
      bADSState := TRUE;
      uiADSStateSeq := 0;
    ELSIF tonADSState.Q THEN
      stSeqCtrlGeneral.eActiveSeqState := E_SEQ_GENERAL.ERROR;
      bADSState := FALSE;
		END_IF
END_CASE
END_ACTION

ACTION A_020_InfluxDBState:
tonInfluxDBState(IN:= NOT bResetInfluxDBStateTimer, PT:= tLifeBitTimeout);
bResetInfluxDBStateTimer := FALSE;
tonInfluxDBState.IN := TRUE;

CASE uiInfluxDBStateSeq OF
  0:
    IF bDBLifeBit AND bAdsConnected THEN
      bResetInfluxDBStateTimer := TRUE;
      bInfluxDBState := TRUE;
      uiInfluxDBStateSeq := 1;
    ELSIF tonInfluxDBState.Q THEN
      stSeqCtrlGeneral.eActiveSeqState := E_SEQ_GENERAL.ERROR;
      bInfluxDBState := FALSE;
		END_IF
  1:
    IF NOT bDBLifeBit AND bAdsConnected THEN
      bResetInfluxDBStateTimer := TRUE;
      bInfluxDBState := TRUE;
      uiInfluxDBStateSeq := 0;
    ELSIF tonInfluxDBState.Q THEN
      stSeqCtrlGeneral.eActiveSeqState := E_SEQ_GENERAL.ERROR;
      bInfluxDBState := FALSE;
		END_IF
END_CASE
END_ACTION

METHOD FB_init : BOOL
VAR_INPUT
	bInitRetains : BOOL; // if TRUE, the retain variables are initialized (warm start / cold start)
	bInCopyCode : BOOL;  // if TRUE, the instance afterwards gets moved into the copy code (online change)
  
  itfOpMode:											                        I_OP_MODE;  
  itfEventLogger:                                         I_EVENT_LOGGER;
END_VAR
THIS^.itfOpMode := itfOpMode;
THIS^.itfEventLogger := itfEventLogger;
END_METHOD

METHOD M_BucketExistCheck : BOOL
VAR_INPUT
	(* Name of the table that is to be read.*)
	sBucketName	: Tc2_System.T_MaxString;
END_VAR
VAR_OUTPUT
	(* Result*)
	bResult	: BOOL;
END_VAR
// Output
bResult := THIS^.bResult;

M_BucketExistCheck := THIS^.stSeqCtrlGeneral.eActiveSeqState = E_SEQ_GENERAL.DONE;

// Input
THIS^.sBucketName := sBucketName;

// General
IF THIS^.stSeqCtrlGeneral.eActiveSeqState = E_SEQ_GENERAL.READY THEN
  THIS^.eNextSeq := E_SEQ_DATABASE.BUCKET_EXIST_CHECK;
  THIS^.stSeqCtrlGeneral.eActiveSeqState := E_SEQ_GENERAL.EXECUTE;
END_IF
END_METHOD

METHOD M_ClearMeasurement : BOOL
VAR_INPUT
	(* Bucket name*)
	sBucketName	: Tc2_System.T_MaxString;
	(* Name of the measure to clear*)
	sMeasurementName	: Tc2_System.T_MaxString;
	(* From date time (Range)*)
	dtFrom	: DATE_AND_TIME;
	(* To date time (Range)*)
	dtTo	: DATE_AND_TIME;
END_VAR
VAR_OUTPUT
	(* Result*)
	bResult	: BOOL;
END_VAR
// Output
bResult := THIS^.bResult;

M_ClearMeasurement := THIS^.stSeqCtrlGeneral.eActiveSeqState = E_SEQ_GENERAL.DONE;

// Input
THIS^.sBucketName := sBucketName;
THIS^.sMeasurementName := sMeasurementName;
THIS^.dtFrom := dtFrom;
THIS^.dtTo := dtTo;

// General
IF THIS^.stSeqCtrlGeneral.eActiveSeqState = E_SEQ_GENERAL.READY THEN
  THIS^.eNextSeq := E_SEQ_DATABASE.CLEAR_MEASUREMENT;
  THIS^.stSeqCtrlGeneral.eActiveSeqState := E_SEQ_GENERAL.EXECUTE;
END_IF
END_METHOD

METHOD M_DeleteAllMeasurements : BOOL
VAR_INPUT
	(* Bucket name*)
	sBucketName	: Tc2_System.T_MaxString;
END_VAR
VAR_OUTPUT
	(* Result*)
	bResult	: BOOL;
END_VAR
// Output
bResult := THIS^.bResult;

M_DeleteAllMeasurements := THIS^.stSeqCtrlGeneral.eActiveSeqState = E_SEQ_GENERAL.DONE;

// Input
THIS^.sBucketName := sBucketName;

// General
IF THIS^.stSeqCtrlGeneral.eActiveSeqState = E_SEQ_GENERAL.READY THEN
  THIS^.eNextSeq := E_SEQ_DATABASE.DELETE_ALL_MEASUREMENTS;
  THIS^.stSeqCtrlGeneral.eActiveSeqState := E_SEQ_GENERAL.EXECUTE;
END_IF
END_METHOD

METHOD M_DeleteField : BOOL
VAR_INPUT
	(* Bucket name*)
	sBucketName	: Tc2_System.T_MaxString;
	(* Measurement Name*)
	sMeasurementName	: Tc2_System.T_MaxString;
	(* Tag Name*)
	sTagName	: Tc2_System.T_MaxString;
	(* Field Name*)
	sFieldName	: Tc2_System.T_MaxString;
END_VAR
VAR_OUTPUT
	(* Result*)
	bResult	: BOOL;
END_VAR
// Output
bResult := THIS^.bResult;

M_DeleteField := THIS^.stSeqCtrlGeneral.eActiveSeqState = E_SEQ_GENERAL.DONE;

// Input
THIS^.sBucketName := sBucketName;
THIS^.sMeasurementName := sMeasurementName;
THIS^.sTagName := sTagName;
THIS^.sFieldNameExistCheck := sFieldName;

// General
IF THIS^.stSeqCtrlGeneral.eActiveSeqState = E_SEQ_GENERAL.READY THEN
  THIS^.eNextSeq := E_SEQ_DATABASE.DELETE_FIELD;
  THIS^.stSeqCtrlGeneral.eActiveSeqState := E_SEQ_GENERAL.EXECUTE;
END_IF
END_METHOD

METHOD M_DeleteMeasurement : BOOL
VAR_INPUT
	(* Bucket name*)
	sBucketName	: Tc2_System.T_MaxString;
	(* Name of the measure to delete.*)
	sMeasurementName	: Tc2_System.T_MaxString;
END_VAR
VAR_OUTPUT
	(* Result*)
	bResult	: BOOL;
END_VAR
// Output
bResult := THIS^.bResult;

M_DeleteMeasurement := THIS^.stSeqCtrlGeneral.eActiveSeqState = E_SEQ_GENERAL.DONE;

// Input
THIS^.sBucketName := sBucketName;
THIS^.sMeasurementName := sMeasurementName;

// General
IF THIS^.stSeqCtrlGeneral.eActiveSeqState = E_SEQ_GENERAL.READY THEN
  THIS^.eNextSeq := E_SEQ_DATABASE.DELETE_MEASUREMENT;
  THIS^.stSeqCtrlGeneral.eActiveSeqState := E_SEQ_GENERAL.EXECUTE;
END_IF
END_METHOD

METHOD M_DeleteTag : BOOL
VAR_INPUT
	(* Bucket name*)
	sBucketName	: Tc2_System.T_MaxString;
	(* Measurement Name*)
	sMeasurementName	: Tc2_System.T_MaxString;
	(* Tag Name*)
	sTagName	: Tc2_System.T_MaxString;
END_VAR
VAR_OUTPUT
	(* Result*)
	bResult	: BOOL;
END_VAR
// Output
bResult := THIS^.bResult;

M_DeleteTag := THIS^.stSeqCtrlGeneral.eActiveSeqState = E_SEQ_GENERAL.DONE;

// Input
THIS^.sBucketName := sBucketName;
THIS^.sMeasurementName := sMeasurementName;
THIS^.sTagName := sTagName;

// General
IF THIS^.stSeqCtrlGeneral.eActiveSeqState = E_SEQ_GENERAL.READY THEN
  THIS^.eNextSeq := E_SEQ_DATABASE.DELETE_TAG;
  THIS^.stSeqCtrlGeneral.eActiveSeqState := E_SEQ_GENERAL.EXECUTE;
END_IF
END_METHOD

METHOD M_DeleteTagContentBlock : BOOL
VAR_INPUT
	(* Bucket name*)
	sBucketName	: Tc2_System.T_MaxString;
	(* Measurement Name*)
	sMeasurementName	: Tc2_System.T_MaxString;
	(* Tag Name*)
	sTagName	: Tc2_System.T_MaxString;
	(* Date and time from*)
	dtFrom	: DATE_AND_TIME;
	(* Date and Time to*)
	dtTo	: DATE_AND_TIME;
END_VAR
VAR_OUTPUT
	(* Result*)
	bResult	: BOOL;
END_VAR
// Output
bResult := THIS^.bResult;

M_DeleteTagContentBlock := THIS^.stSeqCtrlGeneral.eActiveSeqState = E_SEQ_GENERAL.DONE;

// Input
THIS^.sBucketName := sBucketName;
THIS^.sMeasurementName := sMeasurementName;
THIS^.sTagName := sTagName;
THIS^.dtFrom := dtFrom;
THIS^.dtTo := dtTo;

// General
IF THIS^.stSeqCtrlGeneral.eActiveSeqState = E_SEQ_GENERAL.READY THEN
  THIS^.eNextSeq := E_SEQ_DATABASE.DELETE_TAG_CONTENT_BLOCK;
  THIS^.stSeqCtrlGeneral.eActiveSeqState := E_SEQ_GENERAL.EXECUTE;
END_IF
END_METHOD

METHOD M_FieldExistCheck : BOOL
VAR_INPUT
	(* Bucket name*)
	sBucketName	: Tc2_System.T_MaxString;
	(* Measurement Name*)
	sMeasurementName	: Tc2_System.T_MaxString;
	(* Tag Name*)
	sTagName	: Tc2_System.T_MaxString;
	(* Field Name*)
	sFieldName	: Tc2_System.T_MaxString;
END_VAR
VAR_OUTPUT
	(* Result*)
	bResult	: BOOL;
END_VAR
// Output
bResult := THIS^.bResult;

M_FieldExistCheck := THIS^.stSeqCtrlGeneral.eActiveSeqState = E_SEQ_GENERAL.DONE;

// Input
THIS^.sBucketName := sBucketName;
THIS^.sMeasurementName := sMeasurementName;
THIS^.sTagName := sTagName;
THIS^.sFieldNameExistCheck := sFieldName;

// General
IF THIS^.stSeqCtrlGeneral.eActiveSeqState = E_SEQ_GENERAL.READY THEN
  THIS^.eNextSeq := E_SEQ_DATABASE.FIELD_EXIST_CHECK;
  THIS^.stSeqCtrlGeneral.eActiveSeqState := E_SEQ_GENERAL.EXECUTE;
END_IF
END_METHOD

METHOD M_GetTotalMeasurements : BOOL
VAR_INPUT
	(* Bucket name*)
	sBucketName	: Tc2_System.T_MaxString;
END_VAR
VAR_OUTPUT
  (* Process success*)
  bResult:    BOOL;
	(* Result value*)
	uiResult:   UINT;
END_VAR
// Output
bResult := THIS^.bResult;
uiResult := THIS^.uiTotalMeasurements;

M_GetTotalMeasurements := THIS^.stSeqCtrlGeneral.eActiveSeqState = E_SEQ_GENERAL.DONE;

// Input
THIS^.sBucketName := sBucketName;

// General
IF THIS^.stSeqCtrlGeneral.eActiveSeqState = E_SEQ_GENERAL.READY THEN
  THIS^.eNextSeq := E_SEQ_DATABASE.GET_TOTAL_MEASUREMENTS;
  THIS^.stSeqCtrlGeneral.eActiveSeqState := E_SEQ_GENERAL.EXECUTE;
END_IF
END_METHOD

METHOD M_MeasurementExistCheck : BOOL
VAR_INPUT
	(* Bucket name*)
	sBucketName	: Tc2_System.T_MaxString;
	(* Name of the table that is to be read.*)
	sMeasurementName	: Tc2_System.T_MaxString;
END_VAR
VAR_OUTPUT
	(* Result*)
	bResult	: BOOL;
END_VAR
// Output
bResult := THIS^.bResult;

M_MeasurementExistCheck := THIS^.stSeqCtrlGeneral.eActiveSeqState = E_SEQ_GENERAL.DONE;

// Input
THIS^.sBucketName := sBucketName;
THIS^.sMeasurementName := sMeasurementName;

// General
IF THIS^.stSeqCtrlGeneral.eActiveSeqState = E_SEQ_GENERAL.READY THEN
  THIS^.eNextSeq := E_SEQ_DATABASE.MEASUREMENT_EXIST_CHECK;
  THIS^.stSeqCtrlGeneral.eActiveSeqState := E_SEQ_GENERAL.EXECUTE;
END_IF
END_METHOD

METHOD M_Reset : BOOL
M_Reset := THIS^.stSeqCtrlGeneral.eActiveSeqState = E_SEQ_GENERAL.DONE;

// General
IF THIS^.stSeqCtrlGeneral.eActiveSeqState = E_SEQ_GENERAL.READY THEN
  THIS^.eNextSeq := E_SEQ_DATABASE.INIT;
  THIS^.stSeqCtrlGeneral.eActiveSeqState := E_SEQ_GENERAL.EXECUTE;
END_IF
END_METHOD

(*=== Method: M_Run  ============================================

 @brief: Here is the global code (Timer, Event, Flange,...)*)
METHOD M_Run
END_METHOD

METHOD M_SetReady : BOOL
VAR_INPUT
END_VAR
M_SetReady := TRUE
              AND THIS^.stSeqCtrlGeneral.eActiveSeqState = E_SEQ_GENERAL.READY
              AND THIS^.eSeq = E_SEQ_DATABASE.BASE;

THIS^.stSeqCtrlGeneral.eActiveSeqState := E_SEQ_GENERAL.READY;
THIS^.eNextSeq := E_SEQ_DATABASE.BASE;
END_METHOD

METHOD M_TagExistCheck : BOOL
VAR_INPUT
	(* Bucket name*)
	sBucketName	: Tc2_System.T_MaxString;
	(* Measurement Name*)
	sMeasurementName	: Tc2_System.T_MaxString;
	(* Tag Name*)
	sTagName	: Tc2_System.T_MaxString;
END_VAR
VAR_OUTPUT
	(* Result*)
	bResult	: BOOL;
END_VAR
// Output
bResult := THIS^.bResult;

M_TagExistCheck := THIS^.stSeqCtrlGeneral.eActiveSeqState = E_SEQ_GENERAL.DONE;

// Input
THIS^.sBucketName := sBucketName;
THIS^.sMeasurementName := sMeasurementName;
THIS^.sTagName := sTagName;

// General
IF THIS^.stSeqCtrlGeneral.eActiveSeqState = E_SEQ_GENERAL.READY THEN
  THIS^.eNextSeq := E_SEQ_DATABASE.TAG_EXIST_CHECK;
  THIS^.stSeqCtrlGeneral.eActiveSeqState := E_SEQ_GENERAL.EXECUTE;
END_IF
END_METHOD

METHOD M_WriteStruct : BOOL
VAR_INPUT
	(* Bucket name*)
	sBucketName:                  T_MaxString;
	(* Name of the table that is to be read.*)
	sMeasurementName:             T_MaxString;
	(* Tag name*)
	sTagName:                     T_MaxString;
  (* Field values list*)
	stFieldValues:                ST_DATABASE_RECORD;
  (* Field struct content (Variable names) *)
  //pFieldStructContent:          POINTER TO ARRAY [0..99] OF T_MaxString;
	(* Field names list: names that appear in the database*)
	//pFieldNames:                  POINTER TO ARRAY [0..99] OF T_MaxString;
END_VAR
VAR_OUTPUT
	(* Result*)
	bResult	: BOOL;
END_VAR
// Output
bResult := THIS^.bResult;

M_WriteStruct := THIS^.stSeqCtrlGeneral.eActiveSeqState = E_SEQ_GENERAL.DONE;

// Input
THIS^.sBucketName := sBucketName;
THIS^.sMeasurementName := sMeasurementName;
THIS^.sTagName := sTagName;
THIS^.stFieldValues := stFieldValues;
//THIS^.pFieldStructContent := pFieldStructContent;
//THIS^.pFieldNames := pFieldNames;



// General
IF THIS^.stSeqCtrlGeneral.eActiveSeqState = E_SEQ_GENERAL.READY THEN
  THIS^.eNextSeq := E_SEQ_DATABASE.WRITE_STRUCT;
  THIS^.stSeqCtrlGeneral.eActiveSeqState := E_SEQ_GENERAL.EXECUTE;
END_IF
END_METHOD

PROPERTY P_ADSLifebit : BOOL
GET
P_ADSLifebit := THIS^.bADSLifeBit;
END_GET
END_PROPERTY

{warning 'Eigenschaftenimplementierung hinzufügen'}
PROPERTY P_ADSState : BOOL
GET
P_ADSState := THIS^.bADSState;
END_GET
END_PROPERTY

PROPERTY P_Connected : BOOL
GET
P_Connected := false;
END_GET
END_PROPERTY

{warning 'Eigenschaftenimplementierung hinzufügen'}
PROPERTY P_Error : BOOL
GET
P_Error := THIS^.stSeqCtrlGeneral.eActiveSeqState = E_SEQ_GENERAL.ERROR;
END_GET
END_PROPERTY

{warning 'Eigenschaftenimplementierung hinzufügen'}
(*=== Property: P_Event  ============================================

 @param [set]: 	Set the Structure "ST_EVENT" from another Object
 @param [get]: 	Return the Structure "ST_EVENT", it contains the actual 
					event of the Object *)
PROPERTY P_Event : GenLib.ST_EVENT
GET
END_GET
SET
END_SET
END_PROPERTY

{warning 'Eigenschaftenimplementierung hinzufügen'}
(*=== Property: P_FullObjectPath  ============================================

 @param [set]: 	Set the Object Path (Clear String of Object)
 @param [get]: 	Return the Objectpath *)
PROPERTY P_FullObjectPath : STRING
GET
P_FullObjectPath:= THIS^.strFullObjectPath;
END_GET
SET
THIS^.strFullObjectPath:=P_FullObjectPath;
END_SET
END_PROPERTY

{warning 'Eigenschaftenimplementierung hinzufügen'}
(*=== Property: P_Global_Ack  ============================================

 @param [set]: 	Set the Bit for Ack from another Object
 @param [get]: 	Return the state of Ack Bit*)
PROPERTY P_Global_Ack : BOOL
GET
END_GET
SET
END_SET
END_PROPERTY

{warning 'Eigenschaftenimplementierung hinzufügen'}
(*=== Property: P_GlobalID  ============================================

 @param [set]: 	-
 @param [get]: 	Return the string of instance path*)
PROPERTY P_GlobalID : STRING
GET
P_GlobalID:= THIS^.strInstancePath;
END_GET
END_PROPERTY

{warning 'Eigenschaftenimplementierung hinzufügen'}
PROPERTY P_InfluxDBLifeBit : BOOL
GET
P_InfluxDBLifeBit := THIS^.bDBLifeBit;
END_GET
END_PROPERTY

PROPERTY P_InfluxDBState : BOOL
GET
P_InfluxDBState := THIS^.bInfluxDBState;
END_GET
END_PROPERTY

END_FUNCTION_BLOCK

// ---- ORGANISATION/GENERAL/POU/F_CreateObjectName.TcPOU
FUNCTION F_CreateObjectName : STRING
VAR_INPUT
	strObjecktPath: STRING;
END_VAR
VAR
	strTemp: STRING;
	i: INT;
END_VAR


strTemp:=strObjecktPath;

FOR i:=1 TO 10 BY 1 DO
	IF FIND(strTemp,'.')>0 THEN
		strTemp:=DELETE(strTemp,FIND(strTemp,'.')+1,0);
	ELSE
		EXIT;
	END_IF
END_FOR

IF left(strTemp,2)='fb' THEN
	strTemp:=DELETE(strTemp,3,0);
END_IF

F_CreateObjectName:=strTemp;

END_FUNCTION

// ---- PROGRAMS/PrgOrg.TcPOU
{attribute 'global_init_slot' := '40010'}
//{warning 'Safety überarbeiten 170119'}
PROGRAM PrgOrg
VAR_INPUT
  bInitOK:                                 BOOL;
END_VAR
VAR
	fbLocalSysTime: 				                    FB_LOC_SYS_TIME;
	//fbEventHandler: 				                    FB_HANDLE_EVENTS_TXT(itfLocSysTime:=fbLocalSysTime, strPath:='C:\Event\Event.csv');
  fbEventLogger:                              FB_EVENT_LOGGER();
	
// Safety IO  
// Input Sensors
  // EL1918 - 8-chanel-digital-input (KF1.2.1)                 		
  fbEStopLeft_Ch1: 						                FB_BINARY_SWITCH(bInNC:=TRUE);
  fbEStopLeft_Ch2: 						                FB_BINARY_SWITCH(bInNC:=TRUE);
  fbEStopRight_Ch1: 						              FB_BINARY_SWITCH(bInNC:=TRUE);
  fbSafetyDoorLeft_Ch1: 						          FB_BINARY_SWITCH(bInNC:=TRUE);
  fbSafetyDoorLeft_Ch2: 						          FB_BINARY_SWITCH(bInNC:=TRUE);
  fbSafetyDoorRight_Ch1: 						          FB_BINARY_SWITCH(bInNC:=TRUE);
  fbSafetyDoorRight_Ch2: 						          FB_BINARY_SWITCH(bInNC:=TRUE);
  // EL1904 - 4-chanel-digital-input (KF1.2.2) 
  fbEStopJog_Ch1: 						                FB_BINARY_SWITCH(bInNC:=TRUE);
  fbEStopJog_Ch2: 						                FB_BINARY_SWITCH(bInNC:=TRUE);
  fbJog_AckBtn_Ch1: 						              FB_BINARY_SWITCH(bInNC:=TRUE);
  fbJog_AckBtb_Ch2: 						              FB_BINARY_SWITCH(bInNC:=TRUE);
  // EL1904 - 4-chanel-digital-input (KF1.2.3) 
  fbJog_KeySwitch: 						                FB_BINARY_SWITCH(bInNC:=TRUE);
  fbEStop_FeedbackCircuit: 						        FB_BINARY_SWITCH(bInNC:=TRUE);
  fbSafetyDoor_FeedbackCircuit: 						  FB_BINARY_SWITCH(bInNC:=TRUE);
  fbJog_FeedbackCircuit: 						          FB_BINARY_SWITCH(bInNC:=TRUE);
  // EL1904 - 4-chanel-digital-input (KF1.2.4) 
  fbServiceDoorLeft_TestClock_Ch1: 						FB_BINARY_SWITCH(bInNC:=TRUE);
  fbServiceDoorLeft_TestClock_Ch2: 						FB_BINARY_SWITCH(bInNC:=TRUE);
  fbServiceDoorRight_TestClock_Ch1: 					FB_BINARY_SWITCH(bInNC:=TRUE);
  fbServiceDoorRight_TestClock_Ch2: 					FB_BINARY_SWITCH(bInNC:=TRUE);
  // EL1904 - 4-chanel-digital-input (KF1.2.5) 
  fbCounterCyl1_JogValvePos: 						      FB_BINARY_SWITCH(bInNC:=TRUE);
  fbCounterCyl2_JogValvePos: 						      FB_BINARY_SWITCH(bInNC:=TRUE);
  fbCounterCyl3_JogValvePos: 						      FB_BINARY_SWITCH(bInNC:=TRUE);
  fbCounterCyl4_JogValvePos: 						      FB_BINARY_SWITCH(bInNC:=TRUE);
  
  /////////////////////////////////////////
  // EL1018 - 8-chanel-digital-input (KF1.5.0)
  fbPowerAdapter24V_Hydraulics_Ok:                FB_BINARY_SWITCH(bInNC:= FALSE);
  fbSelectivityModules_Ok:                        FB_BINARY_SWITCH(bInNC:= FALSE);
  fbCircuitBreaker_Ok:                            FB_BINARY_SWITCH(bInNC:= FALSE);
  fbCabinetTemperature_Ok:                        FB_BINARY_SWITCH(bInNC:= FALSE);
  // EL1018 - 8-chanel-digital-input (KF1.5.1)
  fbUnitConnector1_Contacted:                     FB_BINARY_SWITCH(bInNC:= FALSE);
  fbUnitConnector2_Contacted:                     FB_BINARY_SWITCH(bInNC:= FALSE);
  fbUnitConnector3_Contacted:                     FB_BINARY_SWITCH(bInNC:= FALSE);
  fbUnitConnector4_Contacted:                     FB_BINARY_SWITCH(bInNC:= FALSE);
  fbLiquiphant_TestBench_Triggered:               FB_BINARY_SWITCH(bInNC:= FALSE);
  fbLiquiphant_ValveBlocks_Triggered:             FB_BINARY_SWITCH(bInNC:= FALSE);
	
  // Other                   			
	fbOpMode:							                      FB_OP_MODE_PAUSE( itfEventLogger:= fbEventLogger, 
	                                                              itfPowerAdapter24V_Hydraulics_Ok:= fbPowerAdapter24V_Hydraulics_Ok, 
	                                                              itfSelectivityModules_Ok:= fbSelectivityModules_Ok, 
	                                                              itfCircuitBreaker_Ok:= fbCircuitBreaker_Ok, 
	                                                              itfCabinetTemperature_Ok:= fbCabinetTemperature_Ok, 
	                                                              itfUnitConnector1_Contacted:= fbUnitConnector1_Contacted, 
	                                                              itfUnitConnector2_Contacted:= fbUnitConnector2_Contacted, 
	                                                              itfUnitConnector3_Contacted:= fbUnitConnector3_Contacted, 
	                                                              itfUnitConnector4_Contacted:= fbUnitConnector4_Contacted, 
	                                                              itfLiquiphant_TestBench_Triggered:= fbLiquiphant_TestBench_Triggered, 
	                                                              itfLiquiphant_ValveBlocks_Triggered:= fbLiquiphant_ValveBlocks_Triggered,
                                                                itfFromSafety_EStop_Ok:= fbFromSafety_EStop_Ok,
                                                                itfFromSafety_SafetyDoor_Ok:= fbFromSafety_SafetyDoor_Ok,
                                                                itfFromSafety_KeySwitch_JogPos:= fbFromSafety_KeySwitch_JogPos,
                                                                itfFromSafety_EStopLeft_Ok:= fbFromSafety_EStopLeft_Ok,
                                                                itfFromSafety_EStopRight_Ok:= fbFromSafety_EStopRight_Ok,
                                                                itfFromSafety_EStopJog_Ok:= fbFromSafety_EStopJog_Ok,
                                                                itfFromSafety_SafetyDoorLeft_Ok:= fbFromSafety_SafetyDoorLeft_Ok,
                                                                itfFromSafety_SafetyDoorRight_Ok:= fbFromSafety_SafetyDoorRight_Ok,
                                                                itfFromSafety_ServiceDoorLeft_Ok:= fbFromSafety_ServiceDoorLeft_Ok,
                                                                itfFromSafety_ServiceDoorRight_Ok:= fbFromSafety_ServiceDoorRight_Ok,
                                                                itfFromSafety_JogAckBtn_Pressed:= fbFromSafety_JogAckBtn_Pressed,
                                                                itfFromSafety_StateServiceValve1:= fbFromSafety_StateServiceValve1,
                                                                itfFromSafety_StateServiceValve2:= fbFromSafety_StateServiceValve2,
                                                                itfFromSafety_StateServiceValve3:= fbFromSafety_StateServiceValve3,
                                                                itfFromSafety_StateServiceValve4:= fbFromSafety_StateServiceValve4,
                                                                itfFromSafety_ServiceMode_Ok:= fbFromSafety_ServiceMode_Ok,
                                                                itfFromSafety_ServiceValves_Ok:= fbFromSafety_ServiceValves_Ok);
  fbTrafficLight:                             FB_TrafficLight(itfLightGreen:= PrgStation.fbTrafficLight_Green, 
                                                              itfLightYellow:= PrgStation.fbTrafficLight_Yellow, 
                                                              itfLightRed:= PrgStation.fbTrafficLight_Red, 
                                                              itfBeep:= PrgStation.fbTrafficLight_Beep);
	fbUserMng: 							                    FB_USER_MANAGER_OLD;

	
  // From Safety
	tonInitQuit:						                    TON;
	
	fbErrorACK: 						                    FB_BINARY_OUTPUT;
	fbSafetyRun: 						                    FB_BINARY_OUTPUT;
	fbSafetyRestart:										        FB_BINARY_OUTPUT;
	fbLockDoor:												          FB_BINARY_OUTPUT;
               					
	fbComErr:							                      FB_BINARY_SWITCH(bInNC:= FALSE);
	fbErr:								                      FB_BINARY_SWITCH(bInNC:= FALSE);
	fbIn:								                        FB_BINARY_SWITCH(bInNC:= FALSE);
	
	tpErrAck:							                      TP;           	
	tpQuit: 							                      TP;
	fTrigAck:							                      F_TRIG;
	tpTrigAck:							                    TP;
  tonAck:                                     TON;
  bAck:                                       BOOL;
  uiAckSeq:                                   UINT := 0;
  
  // From safety
  fbFromSafety_EStop_Ok:                      FB_BINARY_SWITCH(bInNC:= FALSE);
  fbFromSafety_SafetyDoor_Ok:                 FB_BINARY_SWITCH(bInNC:= FALSE);
  fbFromSafety_KeySwitch_JogPos:              FB_BINARY_SWITCH(bInNC:= FALSE);
  fbFromSafety_EStopLeft_Ok:                  FB_BINARY_SWITCH(bInNC:= FALSE);
  fbFromSafety_EStopRight_Ok:                 FB_BINARY_SWITCH(bInNC:= FALSE);
  fbFromSafety_EStopJog_Ok:                   FB_BINARY_SWITCH(bInNC:= FALSE);
  fbFromSafety_SafetyDoorLeft_Ok:             FB_BINARY_SWITCH(bInNC:= FALSE);
  fbFromSafety_SafetyDoorRight_Ok:            FB_BINARY_SWITCH(bInNC:= FALSE);
  fbFromSafety_ServiceDoorLeft_Ok:            FB_BINARY_SWITCH(bInNC:= FALSE);
  fbFromSafety_ServiceDoorRight_Ok:           FB_BINARY_SWITCH(bInNC:= FALSE);
  fbFromSafety_JogAckBtn_Pressed:             FB_BINARY_SWITCH(bInNC:= FALSE);
  fbFromSafety_StateServiceValve1:            FB_BINARY_SWITCH(bInNC:= FALSE);
  fbFromSafety_StateServiceValve2:            FB_BINARY_SWITCH(bInNC:= FALSE);
  fbFromSafety_StateServiceValve3:            FB_BINARY_SWITCH(bInNC:= FALSE);
  fbFromSafety_StateServiceValve4:            FB_BINARY_SWITCH(bInNC:= FALSE);
  fbFromSafety_ServiceMode_Ok:                FB_BINARY_SWITCH(bInNC:= FALSE);
  fbFromSafety_ServiceValves_Ok:              FB_BINARY_SWITCH(bInNC:= FALSE);
END_VAR
VAR
  iOPModeStateInfo:                           INT;
  bStartSafety:                               BOOL;
END_VAR

(* Actions *)
A_000_FBs();
A_010_Init();
A_020_Ack();
A_030_TrafficLight();
A_040_OPMode();

ACTION A_000_FBs:
(* FBs *)
fbOpMode();
fbEventLogger();
fbUserMng();
fbTrafficLight();
END_ACTION

ACTION A_010_Init:

END_ACTION

ACTION A_020_Ack:
IF NOT fbSafetyRun.P_State THEN
  fbSafetyRun.M_Set();
END_IF

IF bAck THEN
  CASE uiAckSeq OF
    0:
      fbErrorACK.M_Set();
      uiAckSeq := 1;
    1:
      tonAck(IN:= NOT tonAck.Q, PT:= T#100MS);
      IF tonAck.Q THEN
        fbErrorACK.M_Reset();
        uiAckSeq := 2;
	    END_IF
    2:
      fbSafetyRestart.M_Set();
      uiAckSeq := 3;
    3:
      tonAck(IN:= NOT tonAck.Q, PT:= T#1S);
      IF tonAck.Q THEN
        fbSafetyRestart.M_Reset();
        uiAckSeq := 0;
        bAck := FALSE;
	    END_IF
	END_CASE
END_IF
END_ACTION

ACTION A_030_TrafficLight:
iOPModeStateInfo := fbOpMode.P_OP_MODE_STATE;

CASE fbOpMode.P_OP_MODE_STATE OF
  OP_MODE.AUTO:
    fbTrafficLight.M_Green(bEnable:= TRUE, uiBlinkFrequency:= 0, bResetOther:= TRUE);
  OP_MODE.INIT, OP_MODE.INIT_OK:
    fbTrafficLight.M_Yellow(bEnable:= TRUE, uiBlinkFrequency:= 0, bResetOther:= TRUE);
  OP_MODE.MANUAL:
    fbTrafficLight.M_Multicolor(bGreen:= TRUE, bYellow:= TRUE, bRed:= FALSE, uiBlinkFrequency:= 0);
  OP_MODE.CONTROL_ON:
    fbTrafficLight.M_Yellow(bEnable:= TRUE, uiBlinkFrequency:= 1, bResetOther:= TRUE);
  OP_MODE.AUTO_TEMPORARY, OP_MODE.RESET_TEMPORARY:
    fbTrafficLight.M_Multicolor(bGreen:= TRUE, bYellow:= TRUE, bRed:= FALSE, uiBlinkFrequency:= 1);
  OP_MODE.MACHINE_ERROR:
    fbTrafficLight.M_Red(bEnable:= TRUE, uiBlinkFrequency:= 1, bResetOther:= TRUE);
  OP_MODE.MANUAL_TEMPORARY:
    fbTrafficLight.M_Multicolor(bGreen:= TRUE, bYellow:= TRUE, bRed:= FALSE, uiBlinkFrequency:= 1);
  OP_MODE.SAFETY_STOP, OP_MODE.STOP:
    fbTrafficLight.M_Red(bEnable:= TRUE, uiBlinkFrequency:= 0, bResetOther:= TRUE);
END_CASE
END_ACTION

ACTION A_040_OPMode:
(* OP Mode *)
fbOpMode.P_INIT_OK := bInitOK;

IF fbFromSafety_KeySwitch_JogPos.P_Active AND fbLockDoor.P_State THEN
  fbLockDoor.M_Reset();
END_IF
END_ACTION

END_PROGRAM

// ---- ORGANISATION/EVENT_LOGGER/POUs/FB_EVENT_LOGGER.TcPOU
FUNCTION_BLOCK FB_EVENT_LOGGER IMPLEMENTS I_EVENT_LOGGER
VAR
  fbAlarm:                        FB_TcAlarm;
  fbMessage:                      FB_TcMessage;
  bError:                         BOOL;
  bInfo:                          BOOL;
  bWarning:                       BOOL;
  uiSeq:                          ARRAY [1..3] OF UINT := [0, 0, 0];
  udiID:                          UDINT;
	sMsg:                           T_MaxString;
  bWithConfirmation:              BOOL;
END_VAR

IF bInfo THEN
  CASE uiSeq[1] OF
    0:
      fbMessage.CreateEx(TC_EVENTS.Info.IndividualInfoMsg, 0);
      uiSeq[1] := 1;
    1:
      fbMessage.ipArguments.Clear().AddDInt(udiID).AddString(sMsg);
      fbMessage.Send(0);
      uiSeq[1] := 2;
    2:
      bInfo := FALSE;
      uiSeq[1] := 0;
	END_CASE
END_IF

IF bWarning THEN
  CASE uiSeq[2] OF
    0:
      fbMessage.CreateEx(TC_EVENTS.Warnings.IndividualWarningMsg, 0);
      uiSeq[2] := 1;
    1:
      fbMessage.ipArguments.Clear().AddDInt(udiID).AddString(sMsg);
      fbMessage.Send(0);
      uiSeq[2] := 2;
    2:
      bWarning := FALSE;
      uiSeq[2] := 0;
	END_CASE
END_IF

IF bError THEN
  CASE uiSeq[3] OF
    0:
      fbAlarm.CreateEx(TC_EVENTS.Errors.IndividualErrMsg, bWithConfirmation, 0);
      uiSeq[3] := 1;
    1:
      fbAlarm.ipArguments.Clear().AddDInt(udiID).AddString(sMsg);
      fbAlarm.Raise(0);
      uiSeq[3] := 2;
    2:
      bError := FALSE;
      uiSeq[3] := 0;
	END_CASE
END_IF

METHOD M_ErrorMsg : BOOL
VAR_INPUT
	udiID:                        UDINT;
	sMsg:                         T_MaxString;
  bWithConfirmation:            BOOL;
END_VAR
M_ErrorMsg := THIS^.uiSeq[3] = 2;

// Assign input
THIS^.udiID := udiID;
THIS^.sMsg := sMsg;
THIS^.bWithConfirmation := bWithConfirmation;

THIS^.bError := TRUE;
END_METHOD

METHOD M_InfoMsg : BOOL
VAR_INPUT
	udiID	: UDINT;
	sMsg	: Tc2_System.T_MaxString;
END_VAR
M_InfoMsg := THIS^.uiSeq[1] = 2;

// Assign input
THIS^.udiID := udiID;
THIS^.sMsg := sMsg;

THIS^.bInfo := TRUE;
END_METHOD

{warning 'Methodenimplementierung hinzufügen'}
(*=== Method: M_Run  ============================================

 @brief: Here is the global code (Timer, Event, Flange,...)*)
METHOD M_Run
END_METHOD

METHOD M_WarningMsg : BOOL
VAR_INPUT
	udiID	: UDINT;
	sMsg	: Tc2_System.T_MaxString;
END_VAR
M_WarningMsg := THIS^.uiSeq[2] = 2;

// Assign input
THIS^.udiID := udiID;
THIS^.sMsg := sMsg;

THIS^.bWarning := TRUE;
END_METHOD

{warning 'Eigenschaftenimplementierung hinzufügen'}
(*=== Property: P_Event  ============================================

 @param [set]: 	Set the Structure "ST_EVENT" from another Object
 @param [get]: 	Return the Structure "ST_EVENT", it contains the actual 
					event of the Object *)
PROPERTY P_Event : GenLib.ST_EVENT
GET
END_GET
SET
END_SET
END_PROPERTY

{warning 'Eigenschaftenimplementierung hinzufügen'}
(*=== Property: P_FullObjectPath  ============================================

 @param [set]: 	Set the Object Path (Clear String of Object)
 @param [get]: 	Return the Objectpath *)
PROPERTY P_FullObjectPath : STRING
GET
END_GET
SET
END_SET
END_PROPERTY

{warning 'Eigenschaftenimplementierung hinzufügen'}
(*=== Property: P_Global_Ack  ============================================

 @param [set]: 	Set the Bit for Ack from another Object
 @param [get]: 	Return the state of Ack Bit*)
PROPERTY P_Global_Ack : BOOL
GET
END_GET
SET
END_SET
END_PROPERTY

{warning 'Eigenschaftenimplementierung hinzufügen'}
(*=== Property: P_GlobalID  ============================================

 @param [set]: 	-
 @param [get]: 	Return the string of instance path*)
PROPERTY P_GlobalID : STRING
GET
END_GET
END_PROPERTY

END_FUNCTION_BLOCK

// ---- ORGANISATION/OP_MODE/POU/FB_OP_MODE_PAUSE.TcPOU
FUNCTION_BLOCK FB_OP_MODE_PAUSE IMPLEMENTS I_OP_MODE_PAUSE

VAR
	bAutomatic:                                      BOOL;
	bDebug:                                          BOOL;
	bManual:                                         BOOL;
	bReset:                                          BOOL;
	bInitOK:                                         BOOL;
	bInitOKToState:                                  BOOL;
	btemporay_Automatic:                             BOOL;
	btemporay_Debug:                                 BOOL;
	btemporay_Manual:                                BOOL;
	btemporay_Reset:                                 BOOL;
	bMachineStateOK:                                 BOOL;
	bControlOn:                                      BOOL;
  bAllConnectorsContacted:                         BOOL;
  bTemperatureOk:                                  BOOL;
  bLiquiphantStateOk:                              BOOL;
	bEmergancyStop:                                  BOOL;
	bFatalError:                                     BOOL;
	bPauseActivate:                                  BOOL;
	bInPause:                                        BOOL;
	bInPauseTemp:                                    BOOL;
	bStartAfterPause:                                BOOL;
  bServiceModeActive:                              BOOL;
  bStop:                                           BOOL;
	
	fbBlink:                                         FB_Blink;
	bBlinkPause:                                     BOOL;
	tonInitOK:                                       Tc2_Standard.TON;
  
  // FB_init
  itfEventLogger:                                  I_EVENT_LOGGER;
  itfPowerAdapter24V_Hydraulics_Ok:                I_BINARY_SWITCH;
  itfSelectivityModules_Ok:                        I_BINARY_SWITCH;
  itfCircuitBreaker_Ok:                            I_BINARY_SWITCH;
  itfCabinetTemperature_Ok:                        I_BINARY_SWITCH;
  itfUnitConnector1_Contacted:                     I_BINARY_SWITCH;
  itfUnitConnector2_Contacted:                     I_BINARY_SWITCH;
  itfUnitConnector3_Contacted:                     I_BINARY_SWITCH;
  itfUnitConnector4_Contacted:                     I_BINARY_SWITCH;
  itfLiquiphant_TestBench_Triggered:               I_BINARY_SWITCH;
  itfLiquiphant_ValveBlocks_Triggered:             I_BINARY_SWITCH;
  itfFromSafety_EStop_Ok:                          I_BINARY_SWITCH;
  itfFromSafety_SafetyDoor_Ok:                     I_BINARY_SWITCH;
  itfFromSafety_KeySwitch_JogPos:                  I_BINARY_SWITCH;
  itfFromSafety_EStopLeft_Ok:                      I_BINARY_SWITCH;
  itfFromSafety_EStopRight_Ok:                     I_BINARY_SWITCH;
  itfFromSafety_EStopJog_Ok:                       I_BINARY_SWITCH;
  itfFromSafety_SafetyDoorLeft_Ok:                 I_BINARY_SWITCH;
  itfFromSafety_SafetyDoorRight_Ok:                I_BINARY_SWITCH;
  itfFromSafety_ServiceDoorLeft_Ok:                I_BINARY_SWITCH;
  itfFromSafety_ServiceDoorRight_Ok:               I_BINARY_SWITCH;
  itfFromSafety_JogAckBtn_Pressed:                 I_BINARY_SWITCH;
  itfFromSafety_StateServiceValve1:                I_BINARY_SWITCH;
  itfFromSafety_StateServiceValve2:                I_BINARY_SWITCH;
  itfFromSafety_StateServiceValve3:                I_BINARY_SWITCH;
  itfFromSafety_StateServiceValve4:                I_BINARY_SWITCH;
  itfFromSafety_ServiceMode_Ok:                    I_BINARY_SWITCH;
  itfFromSafety_ServiceValves_Ok:                  I_BINARY_SWITCH;
END_VAR


//Check the Machine State
bMachineStateOK := bControlOn 
                   AND bTemperatureOk
                   AND bAllConnectorsContacted
                   AND bLiquiphantStateOk;
bControlOn := itfPowerAdapter24V_Hydraulics_Ok.P_Active
              AND itfSelectivityModules_Ok.P_Active
              AND itfCircuitBreaker_Ok.P_Active
              AND itfFromSafety_EStop_Ok.P_Active;
bTemperatureOk := itfCabinetTemperature_Ok.P_Active;
bAllConnectorsContacted := itfUnitConnector1_Contacted.P_Active
                           AND itfUnitConnector2_Contacted.P_Active
                           AND itfUnitConnector3_Contacted.P_Active
                           AND itfUnitConnector4_Contacted.P_Active;
bLiquiphantStateOk := NOT itfLiquiphant_TestBench_Triggered.P_Active
                      AND NOT itfLiquiphant_ValveBlocks_Triggered.P_Active;
bEmergancyStop := NOT bMachineStateOK;
	
tonInitOK(IN:= bInitOK AND bReset AND bMachineStateOK, PT:= T#100MS);

METHOD FB_init : BOOL
VAR_INPUT
	bInitRetains : BOOL; // if TRUE, the retain variables are initialized (warm start / cold start)
	bInCopyCode : BOOL;  // if TRUE, the instance afterwards gets moved into the copy code (online change)
  
	itfEventLogger:                                  I_EVENT_LOGGER;
	itfPowerAdapter24V_Hydraulics_Ok:                I_BINARY_SWITCH;
  itfSelectivityModules_Ok:                        I_BINARY_SWITCH;
  itfCircuitBreaker_Ok:                            I_BINARY_SWITCH;
  itfCabinetTemperature_Ok:                        I_BINARY_SWITCH;
  itfUnitConnector1_Contacted:                     I_BINARY_SWITCH;
  itfUnitConnector2_Contacted:                     I_BINARY_SWITCH;
  itfUnitConnector3_Contacted:                     I_BINARY_SWITCH;
  itfUnitConnector4_Contacted:                     I_BINARY_SWITCH;
  itfLiquiphant_TestBench_Triggered:               I_BINARY_SWITCH;
  itfLiquiphant_ValveBlocks_Triggered:             I_BINARY_SWITCH;
  itfFromSafety_EStop_Ok:                          I_BINARY_SWITCH;
  itfFromSafety_SafetyDoor_Ok:                     I_BINARY_SWITCH;
  itfFromSafety_KeySwitch_JogPos:                  I_BINARY_SWITCH;
  itfFromSafety_EStopLeft_Ok:                      I_BINARY_SWITCH;
  itfFromSafety_EStopRight_Ok:                     I_BINARY_SWITCH;
  itfFromSafety_EStopJog_Ok:                       I_BINARY_SWITCH;
  itfFromSafety_SafetyDoorLeft_Ok:                 I_BINARY_SWITCH;
  itfFromSafety_SafetyDoorRight_Ok:                I_BINARY_SWITCH;
  itfFromSafety_ServiceDoorLeft_Ok:                I_BINARY_SWITCH;
  itfFromSafety_ServiceDoorRight_Ok:               I_BINARY_SWITCH;
  itfFromSafety_JogAckBtn_Pressed:                 I_BINARY_SWITCH;
  itfFromSafety_StateServiceValve1:                I_BINARY_SWITCH;
  itfFromSafety_StateServiceValve2:                I_BINARY_SWITCH;
  itfFromSafety_StateServiceValve3:                I_BINARY_SWITCH;
  itfFromSafety_StateServiceValve4:                I_BINARY_SWITCH;
  itfFromSafety_ServiceMode_Ok:                    I_BINARY_SWITCH;
  itfFromSafety_ServiceValves_Ok:                  I_BINARY_SWITCH;
END_VAR
THIS^.itfEventLogger := itfEventLogger;
THIS^.itfPowerAdapter24V_Hydraulics_Ok := itfPowerAdapter24V_Hydraulics_Ok;
THIS^.itfSelectivityModules_Ok := itfSelectivityModules_Ok;
THIS^.itfCircuitBreaker_Ok := itfCircuitBreaker_Ok;
THIS^.itfCabinetTemperature_Ok := itfCabinetTemperature_Ok;
THIS^.itfUnitConnector1_Contacted := itfUnitConnector1_Contacted;
THIS^.itfUnitConnector2_Contacted := itfUnitConnector2_Contacted;
THIS^.itfUnitConnector3_Contacted := itfUnitConnector3_Contacted;
THIS^.itfUnitConnector4_Contacted := itfUnitConnector4_Contacted;
THIS^.itfLiquiphant_TestBench_Triggered := itfLiquiphant_TestBench_Triggered;
THIS^.itfLiquiphant_ValveBlocks_Triggered := itfLiquiphant_ValveBlocks_Triggered;
THIS^.itfFromSafety_EStop_Ok := itfFromSafety_EStop_Ok;
THIS^.itfFromSafety_SafetyDoor_Ok := itfFromSafety_SafetyDoor_Ok;
THIS^.itfFromSafety_KeySwitch_JogPos := itfFromSafety_KeySwitch_JogPos;
THIS^.itfFromSafety_EStopLeft_Ok := itfFromSafety_EStopLeft_Ok;
THIS^.itfFromSafety_EStopRight_Ok := itfFromSafety_EStopRight_Ok;
THIS^.itfFromSafety_EStopJog_Ok := itfFromSafety_EStopJog_Ok;
THIS^.itfFromSafety_SafetyDoorLeft_Ok := itfFromSafety_SafetyDoorLeft_Ok;
THIS^.itfFromSafety_SafetyDoorRight_Ok := itfFromSafety_SafetyDoorRight_Ok;
THIS^.itfFromSafety_ServiceDoorLeft_Ok := itfFromSafety_ServiceDoorLeft_Ok;
THIS^.itfFromSafety_ServiceDoorRight_Ok := itfFromSafety_ServiceDoorRight_Ok;
THIS^.itfFromSafety_JogAckBtn_Pressed := itfFromSafety_JogAckBtn_Pressed;
THIS^.itfFromSafety_StateServiceValve1 := itfFromSafety_StateServiceValve1;
THIS^.itfFromSafety_StateServiceValve2 := itfFromSafety_StateServiceValve2;
THIS^.itfFromSafety_StateServiceValve3 := itfFromSafety_StateServiceValve3;
THIS^.itfFromSafety_StateServiceValve4 := itfFromSafety_StateServiceValve4;
THIS^.itfFromSafety_ServiceMode_Ok := itfFromSafety_ServiceMode_Ok;
THIS^.itfFromSafety_ServiceValves_Ok := itfFromSafety_ServiceValves_Ok;
END_METHOD

METHOD M_AUTOMATIC
M_OP_MODE_OFF();	
IF NOT (THIS^.bAutomatic OR THIS^.bPauseActivate) THEN
	//set Temporary OP Mode
  THIS^.btemporay_Debug		:= FALSE;
	THIS^.btemporay_Manual	:= FALSE;
	THIS^.btemporay_Reset		:= FALSE;
	THIS^.btemporay_Automatic	:= NOT THIS^.btemporay_Automatic;
END_IF
END_METHOD

METHOD M_DEBUG
M_OP_MODE_OFF();
IF NOT THIS^.bDebug THEN
		//set Temporary OP Mode
    THIS^.btemporay_Automatic	:= FALSE;
    THIS^.btemporay_Manual	:= FALSE;
		THIS^.btemporay_Reset		:= FALSE;
		THIS^.bPauseActivate		:= FALSE;
		THIS^.btemporay_Debug		:= NOT THIS^.btemporay_Debug;
END_IF
END_METHOD

METHOD M_MANUAL
M_OP_MODE_OFF();
IF NOT THIS^.bManual  THEN
		//set Temporary OP Mode
    THIS^.btemporay_Automatic	:= FALSE;
		THIS^.btemporay_Debug		:= FALSE;
    THIS^.btemporay_Reset		:= FALSE;
		THIS^.bPauseActivate		:= FALSE;
		THIS^.btemporay_Manual	:= NOT THIS^.btemporay_Manual;
END_IF
END_METHOD

METHOD M_OP_MODE_OFF
//every OP Mode off
THIS^.bAutomatic := FALSE;
THIS^.bDebug := FALSE;
THIS^.bManual := FALSE;
THIS^.bReset := FALSE;
THIS^.btemporay_Automatic	:= FALSE;
THIS^.btemporay_Debug := FALSE;
THIS^.btemporay_Manual := FALSE;
THIS^.btemporay_Reset := FALSE;
THIS^.bPauseActivate := FALSE;
THIS^.bInPause := FALSE;
THIS^.bInPauseTemp := FALSE;
THIS^.bStop := TRUE;
END_METHOD

METHOD M_OP_MODE_ON : BOOL
THIS^.bAutomatic := ((THIS^.btemporay_Automatic OR P_PAUSE_ACTIVATE) AND THIS^.bInitOK) OR (THIS^.bPauseActivate AND NOT THIS^.bInPause);
THIS^.bDebug := THIS^.btemporay_Debug AND THIS^.bInitOK;
THIS^.bManual := THIS^.btemporay_Manual;
THIS^.bReset := THIS^.btemporay_Reset;

THIS^.btemporay_Automatic := FALSE;
THIS^.btemporay_Debug := FALSE;
THIS^.btemporay_Manual := FALSE;
THIS^.btemporay_Reset := FALSE;
THIS^.bStop := FALSE;
THIS^.bInPause := FALSE;
THIS^.bInPauseTemp := FALSE;
THIS^.bPauseActivate := FALSE;
END_METHOD

METHOD M_OP_MODE_TO_PAUSE
IF THIS^.P_OP_MODE_STATE=OP_MODE.AUTO THEN
	THIS^.bPauseActivate:=TRUE;
END_IF
END_METHOD

METHOD M_RESET : BOOL
M_OP_MODE_OFF();
IF NOT THIS^.bReset THEN
	//set Temporary OP Mode
  THIS^.btemporay_Automatic	:= FALSE;
  THIS^.btemporay_Debug := FALSE;
	THIS^.btemporay_Manual := FALSE;
	THIS^.bPauseActivate := FALSE;
	THIS^.btemporay_Reset := NOT THIS^.btemporay_Reset;
END_IF;
END_METHOD


PROPERTY P_CONTROL_ON : BOOL
GET
P_CONTROL_ON := bControlOn;
END_GET
SET
bControlOn := P_CONTROL_ON;
END_SET
END_PROPERTY

PROPERTY P_EMERGANCY_STOP : BOOL
GET
P_EMERGANCY_STOP := bEmergancyStop;
END_GET
SET
bEmergancyStop := P_EMERGANCY_STOP;
END_SET
END_PROPERTY

PROPERTY P_INIT_OK : BOOL
GET
P_INIT_OK := P_OP_MODE_STATE = OP_MODE.INIT_OK;
END_GET
SET
bInitOK := P_INIT_OK;
END_SET
END_PROPERTY

PROPERTY P_OP_MODE_STATE : INT
GET
VAR
	thne: INT;
END_VAR
IF P_CONTROL_ON THEN
	P_OP_MODE_STATE := OP_MODE.CONTROL_ON;
END_IF

//IF itfHandleEvents.P_State >= ENUM_EVENT_TYPE.Rd6_Warning THEN
//	P_OP_MODE_STATE := OP_MODE.MACHINE_ERROR;
//END_IF

IF P_EMERGANCY_STOP THEN
	P_OP_MODE_STATE := OP_MODE.SAFETY_STOP;
END_IF

IF THIS^.bStop THEN
	P_OP_MODE_STATE := OP_MODE.STOP;
END_IF

// OP MODE
IF THIS^.tonInitOK.Q THEN
	P_OP_MODE_STATE := OP_MODE.INIT_OK;
END_IF

IF THIS^.bAutomatic AND THIS^.bMachineStateOK THEN
	IF NOT THIS^.bPauseActivate THEN
		P_OP_MODE_STATE := OP_MODE.AUTO;
	ELSE
		P_OP_MODE_STATE := OP_MODE.PAUSE;	
	END_IF
END_IF;
			
IF THIS^.bDebug AND THIS^.bMachineStateOK THEN
	P_OP_MODE_STATE := OP_MODE.DEBUG;
END_IF

IF THIS^.bManual AND THIS^.bMachineStateOK THEN
	P_OP_MODE_STATE := OP_MODE.MANUAL;
END_IF

IF THIS^.bReset AND NOT THIS^.tonInitOK.Q AND THIS^.bMachineStateOK THEN
	P_OP_MODE_STATE := OP_MODE.INIT;
END_IF

// OP MODE TEMP
IF THIS^.btemporay_Automatic AND THIS^.bMachineStateOK THEN
	P_OP_MODE_STATE := OP_MODE.AUTO_TEMPORARY;
END_IF

IF THIS^.btemporay_Debug AND THIS^.bMachineStateOK THEN
	P_OP_MODE_STATE := OP_MODE.DEBUG_TEMPORARY;
END_IF

IF THIS^.btemporay_Manual	AND THIS^.bMachineStateOK THEN
	P_OP_MODE_STATE := OP_MODE.MANUAL_TEMPORARY;
END_IF

IF THIS^.btemporay_Reset AND THIS^.bMachineStateOK THEN
	P_OP_MODE_STATE := OP_MODE.RESET_TEMPORARY;
END_IF

IF THIS^.bMachineStateOK AND THIS^.bInPause THEN
	P_OP_MODE_STATE := OP_MODE.AUTO_TEMPORARY;
END_IF
END_GET
END_PROPERTY

PROPERTY P_PAUSE_ACTIVATE : BOOL
GET
P_PAUSE_ACTIVATE := THIS^.bPauseActivate;
END_GET
END_PROPERTY

{warning 'Eigenschaftenimplementierung hinzufügen'}
PROPERTY P_QUIT : BOOL
GET
END_GET
END_PROPERTY

END_FUNCTION_BLOCK

// ---- MODULE/TRAFFIC_LIGHT/POUs/FB_TrafficLight.TcPOU
FUNCTION_BLOCK FB_TrafficLight IMPLEMENTS I_TrafficLight
VAR	// Input aus FB_init
	itfLightGreen:			            I_BINARY_OUTPUT;
	itfLightYellow:			            I_BINARY_OUTPUT;
	itfLightRed:			              I_BINARY_OUTPUT;
	itfBeep:				                I_BINARY_OUTPUT;
END_VAR
VAR	// Method input variables
	bEnable_Green:			            BOOL;
	bEnable_Yellow:			            BOOL;
	bEnable_Red:			              BOOL;
	bEnable_Beep:			              BOOL;
	uiBlinkFrequency: 		          ARRAY [1..4] OF UINT;
	bResetOther:			              ARRAY [1..3] OF BOOL;
END_VAR
VAR	// Trigger
	bTrigger_Green:			            BOOL;
	bTrigger_Yellow:		            BOOL;
	bTrigger_Red:			              BOOL;
	bTrigger_Beep:			            BOOL;
	bTrigger_Multicolor:	          BOOL;
END_VAR
VAR
	uiSeq:					                ARRAY [1..4] OF UINT := [0,0,0,0];
	tonFreq:				                ARRAY [1..4] OF TON;
	tFreq:					                ARRAY [1..4] OF TIME;
	bBlink_Green:			              BOOL;
	bBlink_Yellow:			            BOOL;
	bBlink_Red:				              BOOL;
	bBlink_Beep:			              BOOL;
END_VAR

(* Sequences *)
_m_Seq010_Green();
_m_Seq020_Yellow();
_m_Seq030_Red();
_m_Seq040_Beep();

METHOD PRIVATE _m_Seq010_Green
VAR_INPUT
END_VAR
bEnable_Green := uiBlinkFrequency[1] <= 0 
				 AND bTrigger_Green
				 AND NOT bResetOther[2]
				 AND NOT bResetOther[3];
bBlink_Green := uiBlinkFrequency[1] > 0 
				AND bTrigger_Green
				AND NOT bResetOther[2]
				AND NOT bResetOther[3];

tFreq[1] := TO_TIME(uiBlinkFrequency[1] * 1000);
tonFreq[1](IN:= NOT tonFreq[1].Q, PT:= tFreq[1]);
IF bBlink_Green THEN
	CASE uiSeq[1] OF
		0:
			bEnable_Green := TRUE;
			IF tonFreq[1].Q THEN
				uiSeq[1] := 1;
			END_IF
		1:
			bEnable_Green := FALSE;
			IF tonFreq[1].Q THEN
				uiSeq[1] := 0;
			END_IF
	END_CASE
END_IF

IF bEnable_Green THEN
  itfLightGreen.M_Set();
ELSE
  itfLightGreen.M_Reset();
END_IF
END_METHOD

METHOD PRIVATE _m_Seq020_Yellow
VAR_INPUT
END_VAR
bEnable_Yellow := uiBlinkFrequency[2] <= 0 
				 AND bTrigger_Yellow
				 AND NOT bResetOther[1]
				 AND NOT bResetOther[3];
bBlink_Yellow := uiBlinkFrequency[2] > 0 
				AND bTrigger_Yellow
				AND NOT bResetOther[1]
				AND NOT bResetOther[3];

tFreq[2] := TO_TIME(uiBlinkFrequency[2] * 1000);
tonFreq[2](IN:= NOT tonFreq[2].Q, PT:= tFreq[2]);
IF bBlink_Yellow THEN
	CASE uiSeq[2] OF
		0:
			bEnable_Yellow := TRUE;
			IF tonFreq[2].Q THEN
				uiSeq[2] := 1;
			END_IF
		1:
			bEnable_Yellow := FALSE;
			IF tonFreq[2].Q THEN
				uiSeq[2] := 0;
			END_IF
	END_CASE
END_IF

IF bEnable_Yellow THEN
  itfLightYellow.M_Set();
ELSE
  itfLightYellow.M_Reset();
END_IF
END_METHOD

METHOD PRIVATE _m_Seq030_Red
VAR_INPUT
END_VAR
bEnable_Red := uiBlinkFrequency[3] <= 0 
				 AND bTrigger_Red
				 AND NOT bResetOther[1]
				 AND NOT bResetOther[2];
bBlink_Red := uiBlinkFrequency[3] > 0 
				AND bTrigger_Red
				AND NOT bResetOther[1]
				AND NOT bResetOther[2];

tFreq[3] := TO_TIME(uiBlinkFrequency[3] * 1000);
tonFreq[3](IN:= NOT tonFreq[3].Q, PT:= tFreq[3]);
IF bBlink_Red THEN
	CASE uiSeq[3] OF
		0:
			bEnable_Red := TRUE;
			IF tonFreq[3].Q THEN
				uiSeq[3] := 1;
			END_IF
		1:
			bEnable_Red := FALSE;
			IF tonFreq[3].Q THEN
				uiSeq[3] := 0;
			END_IF
	END_CASE
END_IF

IF bEnable_Red THEN
  itfLightRed.M_Set();
ELSE
  itfLightRed.M_Reset();
END_IF
END_METHOD

METHOD PRIVATE _m_Seq040_Beep
VAR_INPUT
END_VAR
bEnable_Beep := uiBlinkFrequency[4] <= 0 
				 AND bTrigger_Beep;
bBlink_Beep := uiBlinkFrequency[4] > 0 
				AND bTrigger_Beep;

tFreq[4] := TO_TIME(uiBlinkFrequency[4] * 1000);
tonFreq[4](IN:= NOT tonFreq[4].Q, PT:= tFreq[4]);
IF bBlink_Beep THEN
	CASE uiSeq[4] OF
		0:
			bEnable_Beep := TRUE;
			IF tonFreq[4].Q THEN
				uiSeq[4] := 1;
			END_IF
		1:
			bEnable_Beep := FALSE;
			IF tonFreq[4].Q THEN
				uiSeq[4] := 0;
			END_IF
	END_CASE
END_IF

IF bEnable_Beep THEN
  itfBeep.M_Set();
ELSE
  itfBeep.M_Reset();
END_IF
END_METHOD

METHOD FB_init : BOOL
VAR_INPUT
	bInitRetains:           BOOL; // if TRUE, the retain variables are initialized (warm start / cold start)
	bInCopyCode:            BOOL;  // if TRUE, the instance afterwards gets moved into the copy code (online change)
	
	itfLightGreen:			    I_BINARY_OUTPUT;
	itfLightYellow:			    I_BINARY_OUTPUT;
	itfLightRed:			      I_BINARY_OUTPUT;
	itfBeep:				        I_BINARY_OUTPUT;
END_VAR
THIS^.itfLightGreen := itfLightGreen;
THIS^.itfLightYellow := itfLightYellow;
THIS^.itfLightRed := itfLightRed;
THIS^.itfBeep := itfBeep;
END_METHOD

METHOD M_Beep : BOOL
VAR_INPUT
	(* On/Off signal*)
	bEnable	: BOOL;
	(* Flashing frequency (0 = Permanently On, 1 = 1s alternately, ...)*)
	uiBlinkFrequency	: UINT;
END_VAR
M_Beep := THIS^.bTrigger_Beep = bEnable;

// Assign input
THIS^.bTrigger_Beep := bEnable;
THIS^.uiBlinkFrequency[4] := uiBlinkFrequency;
END_METHOD

METHOD M_Green : BOOL
VAR_INPUT
	(* On/Off light*)
	bEnable: 				BOOL;
	(* Flashing frequency (0 = Permanently On, 1 = 1s alternately, ...)*)
	uiBlinkFrequency: 		UINT;
	(* Reset all colors, before set this color*)
	bResetOther:			BOOL;
END_VAR
M_Green := THIS^.bTrigger_Green = bEnable;

// Assign input
THIS^.bTrigger_Green := bEnable;
THIS^.uiBlinkFrequency[1] := uiBlinkFrequency;
THIS^.bResetOther[1] := bResetOther;
THIS^.bResetOther[2] := THIS^.bResetOther[3] := FALSE;
END_METHOD

METHOD M_Multicolor : BOOL
VAR_INPUT
	(* Enable green*)
	bGreen	: BOOL;
	(* Enable yellow*)
	bYellow	: BOOL;
	(* Enable red*)
	bRed	: BOOL;
	(* Flashing frequency (0 = Permanently On, 1 = 1s alternately, ...)*)
	uiBlinkFrequency	: UINT;
END_VAR
M_Multicolor := THIS^.bTrigger_Red = bGreen;

// Assign input
THIS^.bTrigger_Green := bGreen;
THIS^.bTrigger_Yellow := bYellow;
THIS^.bTrigger_Red := bRed;
THIS^.uiBlinkFrequency[1] := THIS^.uiBlinkFrequency[2] := THIS^.uiBlinkFrequency[3] := uiBlinkFrequency;
THIS^.bResetOther[1] := THIS^.bResetOther[2] := THIS^.bResetOther[3] := FALSE;
END_METHOD

METHOD M_Red : BOOL
VAR_INPUT
	(* On/Off light*)
	bEnable: 				BOOL;
	(* Flashing frequency (0 = Permanently On, 1 = 1s alternately, ...)*)
	uiBlinkFrequency: 		UINT;
	(* Reset all colors, before set this color*)
	bResetOther:			BOOL;
END_VAR
M_Red := THIS^.bTrigger_Red = bEnable;

// Assign input
THIS^.bTrigger_Red := bEnable;
THIS^.uiBlinkFrequency[3] := uiBlinkFrequency;
THIS^.bResetOther[3] := bResetOther;
THIS^.bResetOther[1] := THIS^.bResetOther[2] := FALSE;
END_METHOD

{warning 'Methodenimplementierung hinzufügen'}
METHOD M_Reset : BOOL
END_METHOD

METHOD M_Yellow : BOOL
VAR_INPUT
	(* On/Off light*)
	bEnable: 				BOOL;
	(* Flashing frequency (0 = Permanently On, 1 = 1s alternately, ...)*)
	uiBlinkFrequency: 		UINT;
	(* Reset all colors, before set this color*)
	bResetOther:			BOOL;
END_VAR
M_Yellow := THIS^.bTrigger_Yellow = bEnable;

// Assign input
THIS^.bTrigger_Yellow := bEnable;
THIS^.uiBlinkFrequency[2] := uiBlinkFrequency;
THIS^.bResetOther[2] := bResetOther;
THIS^.bResetOther[1] := THIS^.bResetOther[3] := FALSE;
END_METHOD

PROPERTY P_BeepState : BOOL
GET
P_BeepState := THIS^.itfBeep.P_State;
END_GET
END_PROPERTY

PROPERTY P_GreenState : BOOL
GET
P_GreenState := THIS^.itfLightGreen.P_State;
END_GET
END_PROPERTY

PROPERTY P_RedState : BOOL
GET
P_RedState := THIS^.itfLightRed.P_State;
END_GET
END_PROPERTY

PROPERTY P_YellowState : BOOL
GET
P_YellowState := THIS^.itfLightYellow.P_State;
END_GET
END_PROPERTY

END_FUNCTION_BLOCK

// ---- PROGRAMS/PrgStation.TcPOU
 {attribute 'global_init_slot' := '40020'}
PROGRAM PrgStation
VAR
		
{region 'Step Sequence'}
//Aufruf Hauptschrittkette Ablauf
   uiSeq:                                         UINT := 999;
   uiLastSeq:                                     UINT := 998;
   iLastOPMode:                                   INT := -1;
   bExitSetReadyState:                            BOOL;
   iInfoOPMode:                                   INT;
   bBusyStop:                                     BOOL;
   bBusyInit:                                     BOOL;
{endregion}		
   
{region 'Timer'}
  fbTimerNest1:                                   FB_CLOCK;
  fbTimerNest2:                                   FB_CLOCK;
  fbTimerNest3:                                   FB_CLOCK;
  fbTimerNest4:                                   FB_CLOCK;
{endregion}
   
{region 'IO'}
// Input Sensors
  // EL1018 - 8-chanel-digital-input (KF1.2.0)
  fbSafetyDoorLeft_Contacted:                     FB_BINARY_SWITCH(bInNC:= FALSE);
  fbSafetyDoorRight_Contacted:                    FB_BINARY_SWITCH(bInNC:= FALSE);
  fbJogBtnPos_Pressed:                            FB_BINARY_SWITCH(bInNC:= FALSE);
  fbJogBtnNeg_Pressed:                            FB_BINARY_SWITCH(bInNC:= FALSE); 
  // EL6224 - 4-chanel-communication-interface IO-Link (KF1.8.0)
  diTestCyl1_Distance                             AT %I* : DINT;
  diTestCyl2_Distance                             AT %I* : DINT;
  diTestCyl3_Distance                             AT %I* : DINT;
  diTestCyl4_Distance                             AT %I* : DINT;
  // EL1018 - 8-chanel-digital-input (KF1.10.0)
  fbMotorProtectionSwitch_Unit_Ok:                FB_BINARY_SWITCH(bInNC:= FALSE);
  fbThermalContact_EngineOilCooler:               FB_BINARY_SWITCH(bInNC:= FALSE);
  fbThermalContact_BypassPump:                    FB_BINARY_SWITCH(bInNC:= FALSE);
  fbThermalContact_LowPressurePump:               FB_BINARY_SWITCH(bInNC:= FALSE);     
  // EL1018 - 8-chanel-digital-input (KF1.10.1)
  fbLevelSwitch_AggregateTank1_Out1:              FB_BINARY_SWITCH(bInNC:= FALSE);
  fbLevelSwitch_AggregateTank1_Out2:              FB_BINARY_SWITCH(bInNC:= FALSE);
  fbTemperatureSwitch_AggregateTank1_Out1:        FB_BINARY_SWITCH(bInNC:= FALSE);
  fbTemperatureSwitch_AggregateTank1_Out2:        FB_BINARY_SWITCH(bInNC:= FALSE);
  fbLevelSwitch_AggregateTank2_Out1:              FB_BINARY_SWITCH(bInNC:= FALSE);
  fbLevelSwitch_AggregateTank2_Out2:              FB_BINARY_SWITCH(bInNC:= FALSE);
  fbLevelSwitch_AggregateTank2_Out3:              FB_BINARY_SWITCH(bInNC:= FALSE);
  fbSwitch_AggregateFilter_Dirty:                 FB_BINARY_SWITCH(bInNC:= FALSE);     
  // EL6224 - 4-chanel-communication-interface IO-Link (KF1.13.0)
  iPressureSensor_TestCyl1                        AT %I* : INT;
  iPressureSensor_TestCyl1_A                      AT %I* : INT;
  iPressureSensor_TestCyl1_B                      AT %I* : INT;
  iPressureSensor_CounterCyl1                     AT %I* : INT;
  // EL6224 - 4-chanel-communication-interface IO-Link (KF1.13.1)
  iPressureSensor_LowPressure                     AT %I* : INT;
  iPressureSensor_TestCyl1_BreakPressure_A        AT %I* : INT;
  iPressureSensor_TestCyl1_BreakPressure_B        AT %I* : INT;
  iPressureSensor_TestCyl1_PressureReservoir      AT %I* : INT;
  // EL1018 - 8-chanel-digital-input (KF1.14.0)
  fbMotorProtectionSwitch_TestAxis1_Ok:           FB_BINARY_SWITCH(bInNC:= FALSE);
  fbThermalContact_TestCyl1Pump:                  FB_BINARY_SWITCH(bInNC:= FALSE);
  fbThermalContact_CounterCyl1Pump:               FB_BINARY_SWITCH(bInNC:= FALSE);
  fbShutOffValve_Closed:                          FB_BINARY_SWITCH(bInNC:= FALSE);
  fbShutOffValve_Opened:                          FB_BINARY_SWITCH(bInNC:= FALSE);
  // EL3122 - 2-chanel-analog-input 16Bit (KF1.16.0)
  iTestCyl1_BreakPressureTest_Distance            AT %I* : INT;
  // EL6224 - 4-chanel-communication-interface IO-Link (KF2.2.0)
  iPressureSensor_TestCyl2                        AT %I* : INT;
  iPressureSensor_TestCyl2_A                      AT %I* : INT;
  iPressureSensor_TestCyl2_B                      AT %I* : INT;
  iPressureSensor_CounterCyl2                     AT %I* : INT;
  // EL1018 - 8-chanel-digital-input (KF2.3.0)
  fbMotorProtectionSwitch_TestAxis2_Ok:           FB_BINARY_SWITCH(bInNC:= FALSE);
  fbThermalContact_TestCyl2Pump:                  FB_BINARY_SWITCH(bInNC:= FALSE);
  fbThermalContact_CounterCyl2Pump:               FB_BINARY_SWITCH(bInNC:= FALSE);
  // EL6224 - 4-chanel-communication-interface IO-Link (KF2.11.0)
  iPressureSensor_TestCyl3                        AT %I* : INT;
  iPressureSensor_TestCyl3_A                      AT %I* : INT;
  iPressureSensor_TestCyl3_B                      AT %I* : INT;
  iPressureSensor_CounterCyl3                     AT %I* : INT;
  // EL1018 - 8-chanel-digital-input (KF2.12.0)
  fbMotorProtectionSwitch_TestAxis3_Ok:           FB_BINARY_SWITCH(bInNC:= FALSE);
  fbThermalContact_TestCyl3Pump:                  FB_BINARY_SWITCH(bInNC:= FALSE);
  fbThermalContact_CounterCyl3Pump:               FB_BINARY_SWITCH(bInNC:= FALSE);
  // EL6224 - 4-chanel-communication-interface IO-Link (KF2.20.0)
  iPressureSensor_TestCyl4                        AT %I* : INT;
  iPressureSensor_TestCyl4_A                      AT %I* : INT;
  iPressureSensor_TestCyl4_B                      AT %I* : INT;
  iPressureSensor_CounterCyl4                     AT %I* : INT;
  // EL1018 - 8-chanel-digital-input (KF2.12.0)
  fbMotorProtectionSwitch_TestAxis4_Ok:           FB_BINARY_SWITCH(bInNC:= FALSE);
  fbThermalContact_TestCyl4Pump:                  FB_BINARY_SWITCH(bInNC:= FALSE);
  fbThermalContact_CounterCyl4Pump:               FB_BINARY_SWITCH(bInNC:= FALSE);
   
// Output switches
  // EL2008 - 8-chanel-digital-output (KF1.6.0)
  fbSelectivityModule1_Restart:                   FB_BINARY_OUTPUT;
  fbSelectivityModule2_Restart:                   FB_BINARY_OUTPUT;
  fbSelectivityModule3_Restart:                   FB_BINARY_OUTPUT;
  fbSelectivityModule4_Restart:                   FB_BINARY_OUTPUT;
  // EL2008 - 8-chanel-digital-output (KF1.6.1)
  fbTrafficLight_Red:                             FB_BINARY_OUTPUT;
  fbTrafficLight_Yellow:                          FB_BINARY_OUTPUT;
  fbTrafficLight_Green:                           FB_BINARY_OUTPUT;
  fbTrafficLight_Beep:                            FB_BINARY_OUTPUT;
  // EL2652 - 2-chanel-relay-output (KF1.7.0)
  fbMachineLight:                                 FB_BINARY_OUTPUT;
  // EL2004 - 4-chanel-digital-output (KF1.11.0)
  fbEngine_OilCooler_Start:                       FB_BINARY_OUTPUT; // Hydraulic plan: 02.10
  fbEngine_BypassPump_Start:                      FB_BINARY_OUTPUT; // Hydraulic plan: 02.02
  fbEngine_LowPressurePump_Start:                 FB_BINARY_OUTPUT; // Hydraulic plan: 03.02
  // EL2024 - 4-chanel-digital-output (KF1.11.1)
  fbValve42_LowPressureCircuit_Enable:            FB_BINARY_OUTPUT; // Hydraulic plan: 03.13
  // EL2004 - 4-chanel-digital-output (KF1.15.0)
  fbEngine_TestCyl1Pump_Start:                    FB_BINARY_OUTPUT; // Hydraulic plan: 04.02
  fbEngine_CounterCyl1Pump_Start:                 FB_BINARY_OUTPUT; // Hydraulic plan: 05.02
  // EL4102 - 2-chanel-analog-output (KF1.17.0) 16Bit
  iTestCyl1_Pressure                              AT %Q* : INT;    // Hydraulic plan: 04.13
  iCounterCyl1_Pressure                           AT %Q* : INT;    // Hydraulic plan: 05.43
  // EL4102 - 2-chanel-analog-output (KF1.17.1) 16Bit
  iTestCyl1_LowPressure                           AT %Q* : INT;    // Hydraulic plan: 04.30
  // EL4132 - 2-chanel-analog-output (KF1.17.2) 16Bit
  iValve43_TestCyl1                               AT %Q* : INT;    // Hydraulic plan: 04.48
  // EL4004 - 4-chanel-analog-output (KF1.17.3) 12Bit
  iBNCSocket_TestCyl1_A_Pressure                  AT %Q* : INT;    // Hydraulic plan: 04.58
  iBNCSocket_TestCyl1_B_Pressure                  AT %Q* : INT;    // Hydraulic plan: 04.60
  iBNCSocket_CounterCyl1_Pressure                 AT %Q* : INT;    // Hydraulic plan: 05.44
  iBNCSocket_TestCyl1_Distance                    AT %Q* : INT;    
  // EL4004 - 4-chanel-analog-output (KF1.17.4) 12Bit
  iBNCSocket_TestCyl1_A_BreakPressure             AT %Q* : INT;    // Hydraulic plan: 04.84
  iBNCSocket_TestCyl1_B_BreakPressure             AT %Q* : INT;    // Hydraulic plan: 04.87
  iBNCSocket_TestingCyl1_PressureReservoir        AT %Q* : INT;    // Hydraulic plan: 04.75
  // EL2828 - 8-chanel-digital-output (KF1.19.0)
  fbValve22_TestCyl1_A_Open:                      FB_BINARY_OUTPUT; // Hydraulic plan: 04.46
  fbValve22_TestCyl1_B_Open:                      FB_BINARY_OUTPUT; // Hydraulic plan: 04.46
  fbValve42_CounterCyl1_LowPressureCircuit_Add:   FB_BINARY_OUTPUT; // Hydraulic plan: 03.22
  fbShutOffValve_Close:                           FB_BINARY_OUTPUT; // Hydraulic plan: 04.26
  fbShutOffValve_Open:                            FB_BINARY_OUTPUT; // Hydraulic plan: 04.26
  // EL2828 - 8-chanel-digital-output (KF1.19.1)
  fbValve22_Pump4_Add:                            FB_BINARY_OUTPUT; // Hydraulic plan: 04.50 (Left)
  fbValve22_Pump3_Add:                            FB_BINARY_OUTPUT; // Hydraulic plan: 04.50 (Right)
  fbValve22_Pump2_Add:                            FB_BINARY_OUTPUT; // Hydraulic plan: 04.53
  fbValve22_PressureReservoir_A_Add:              FB_BINARY_OUTPUT; // Hydraulic plan: 04.72 (Left)
  fbValve22_PressureReservoir_B_Add:              FB_BINARY_OUTPUT; // Hydraulic plan: 04.72 (Right)
  fbValve32_SensorBreakPressure_A_Add:            FB_BINARY_OUTPUT; // Hydraulic plan: 04.83
  fbValve32_SensorBreakPressure_B_Add:            FB_BINARY_OUTPUT; // Hydraulic plan: 04.86
  // EL2828 - 8-chanel-digital-output (KF1.21.0)
  fbValve42_CounterCyl1_Bypass_Add:               FB_BINARY_OUTPUT; // Hydraulic plan: 05.13
  fbValve22_CounterCyl1_SinkBlock_Open:           FB_BINARY_OUTPUT; // Hydraulic plan: 05.43
  fbValve22_CounterCyl1_JogMode_Off:              FB_BINARY_OUTPUT; // Hydraulic plan: 05.21
  fbValve43_CounterCyl1_Extend:                   FB_BINARY_OUTPUT; // Hydraulic plan: 05.25
  fbValve43_CounterCyl1_Retract:                  FB_BINARY_OUTPUT; // Hydraulic plan: 05.25
  // EL2004 - 4-chanel-digital-output (KF2.4.0)
  fbEngine_TestCyl2Pump_Start:                    FB_BINARY_OUTPUT; // Hydraulic plan: 06.02
  fbEngine_CounterCyl2Pump_Start:                 FB_BINARY_OUTPUT; // Hydraulic plan: 07.02
  // EL4102 - 2-chanel-analog-output (KF2.5.0) 16Bit
  iTestCyl2_Pressure                              AT %Q* : INT;    // Hydraulic plan: 06.16
  iCounterCyl2_Pressure                           AT %Q* : INT;    // Hydraulic plan: 07.43
  // EL4132 - 2-chanel-analog-output (KF2.5.1) 16Bit
  iValve43_TestCyl2                               AT %Q* : INT;    // Hydraulic plan: 06.38
  // EL4004 - 4-chanel-analog-output (KF2.5.2) 12Bit
  iBNCSocket_TestCyl2_A_Pressure                  AT %Q* : INT;    // Hydraulic plan: 06.42
  iBNCSocket_TestCyl2_B_Pressure                  AT %Q* : INT;    // Hydraulic plan: 06.44
  iBNCSocket_CounterCyl2_Pressure                 AT %Q* : INT;    // Hydraulic plan: 07.44
  iBNCSocket_TestCyl2_Distance                    AT %Q* : INT;
  // EL2828 - 8-chanel-digital-output (KF2.7.0)
  fbValve22_TestCyl2_A_Open:                      FB_BINARY_OUTPUT; // Hydraulic plan: 06.36 (Left)
  fbValve22_TestCyl2_B_Open:                      FB_BINARY_OUTPUT; // Hydraulic plan: 06.36 (Right)
  fbValve42_CounterCyl2_LowPressureCircuit_Add:   FB_BINARY_OUTPUT; // Hydraulic plan: 03.25
  // EL2828 - 8-chanel-digital-output (KF2.9.0)
  fbValve42_CounterCyl2_Bypass_Add:               FB_BINARY_OUTPUT; // Hydraulic plan: 07.13
  fbValve22_CounterCyl2_SinkBlock_Open:           FB_BINARY_OUTPUT; // Hydraulic plan: 07.43
  fbValve22_CounterCyl2_JogMode_Off:              FB_BINARY_OUTPUT; // Hydraulic plan: 07.21
  fbValve43_CounterCyl2_Extend:                   FB_BINARY_OUTPUT; // Hydraulic plan: 07.25
  fbValve43_CounterCyl2_Retract:                  FB_BINARY_OUTPUT; // Hydraulic plan: 07.25
  // EL2004 - 4-chanel-digital-output (KF2.13.0)
  fbEngine_TestCyl3Pump_Start:                    FB_BINARY_OUTPUT; // Hydraulic plan: 08.02
  fbEngine_CounterCyl3Pump_Start:                 FB_BINARY_OUTPUT; // Hydraulic plan: 09.02
  // EL4102 - 2-chanel-analog-output (KF2.14.0) 16Bit
  iTestCyl3_Pressure                              AT %Q* : INT;    // Hydraulic plan: 08.16
  iCounterCyl3_Pressure                           AT %Q* : INT;    // Hydraulic plan: 09.43
  // EL4132 - 2-chanel-analog-output (KF2.14.1) 16Bit
  iValve43_TestCyl3                               AT %Q* : INT;    // Hydraulic plan: 08.38
  // EL4004 - 4-chanel-analog-output (KF2.14.2) 12Bit
  iBNCSocket_TestCyl3_A_Pressure                  AT %Q* : INT;    // Hydraulic plan: 08.42
  iBNCSocket_TestCyl3_B_Pressure                  AT %Q* : INT;    // Hydraulic plan: 08.44
  iBNCSocket_CounterCyl3_Pressure                 AT %Q* : INT;    // Hydraulic plan: 09.44
  iBNCSocket_TestCyl3_Distance                    AT %Q* : INT;
  // EL2828 - 8-chanel-digital-output (KF2.16.0)
  fbValve22_TestCyl3_A_Open:                      FB_BINARY_OUTPUT; // Hydraulic plan: 08.36 (Left)
  fbValve22_TestCyl3_B_Open:                      FB_BINARY_OUTPUT; // Hydraulic plan: 08.36 (Right)
  fbValve42_CounterCyl3_LowPressureCircuit_Add:   FB_BINARY_OUTPUT; // Hydraulic plan: 03.28
  // EL2828 - 8-chanel-digital-output (KF2.18.0)
  fbValve42_CounterCyl3_Bypass_Add:               FB_BINARY_OUTPUT; // Hydraulic plan: 09.13
  fbValve22_CounterCyl3_SinkBlock_Open:           FB_BINARY_OUTPUT; // Hydraulic plan: 09.43
  fbValve22_CounterCyl3_JogMode_Off:              FB_BINARY_OUTPUT; // Hydraulic plan: 09.21
  fbValve43_CounterCyl3_Extend:                   FB_BINARY_OUTPUT; // Hydraulic plan: 09.25
  fbValve43_CounterCyl3_Retract:                  FB_BINARY_OUTPUT; // Hydraulic plan: 09.25
  // EL2004 - 4-chanel-digital-output (KF2.22.0)
  fbEngine_TestCyl4Pump_Start:                    FB_BINARY_OUTPUT; // Hydraulic plan: 10.02
  fbEngine_CounterCyl4Pump_Start:                 FB_BINARY_OUTPUT; // Hydraulic plan: 11.02
  // EL4102 - 2-chanel-analog-output (KF2.23.0) 16Bit
  iTestCyl4_Pressure                              AT %Q* : INT;    // Hydraulic plan: 10.16
  iCounterCyl4_Pressure                           AT %Q* : INT;    // Hydraulic plan: 11.43
  // EL4132 - 2-chanel-analog-output (KF2.23.1) 16Bit
  iValve43_TestCyl4                               AT %Q* : INT;    // Hydraulic plan: 10.38
  // EL4004 - 4-chanel-analog-output (KF2.23.2) 12Bit
  iBNCSocket_TestCyl4_A_Pressure                  AT %Q* : INT;    // Hydraulic plan: 10.42
  iBNCSocket_TestCyl4_B_Pressure                  AT %Q* : INT;    // Hydraulic plan: 10.44
  iBNCSocket_CounterCyl4_Pressure                 AT %Q* : INT;    // Hydraulic plan: 11.44
  iBNCSocket_TestCyl4_Distance                    AT %Q* : INT;
  // EL2828 - 8-chanel-digital-output (KF2.25.0)
  fbValve22_TestCyl4_A_Open:                      FB_BINARY_OUTPUT; // Hydraulic plan: 10.36 (Left)
  fbValve22_TestCyl4_B_Open:                      FB_BINARY_OUTPUT; // Hydraulic plan: 10.36 (Right)
  fbValve42_CounterCyl4_LowPressureCircuit_Add:   FB_BINARY_OUTPUT; // Hydraulic plan: 03.37
  // EL2828 - 8-chanel-digital-output (KF2.27.0)
  fbValve42_CounterCyl4_Bypass_Add:               FB_BINARY_OUTPUT; // Hydraulic plan: 11.13
  fbValve22_CounterCyl4_SinkBlock_Open:           FB_BINARY_OUTPUT; // Hydraulic plan: 11.33
  fbValve22_CounterCyl4_JogMode_Off:              FB_BINARY_OUTPUT; // Hydraulic plan: 11.21
  fbValve43_CounterCyl4_Extend:                   FB_BINARY_OUTPUT; // Hydraulic plan: 11.25
  fbValve43_CounterCyl4_Retract:                  FB_BINARY_OUTPUT; // Hydraulic plan: 11.25
{endregion}
{region 'Converted values'}
  rPressureConverted_TestCyl1:                    REAL;
  rPressureConverted_TestCyl1_A:                  REAL;
  rPressureConverted_TestCyl1_B:                  REAL;
  rPressureConverted_CounterCyl1:                 REAL;
  rPressureConverted_LowPressure:                 REAL;
  rPressureConverted_TestCyl1_BreakPressure_A:    REAL;
  rPressureConverted_TestCyl1_BreakPressure_B:    REAL;
  rPressureConverted_TestCyl1_PressureReservoir:  REAL;
  rPressureConverted_TestCyl2:                    REAL;
  rPressureConverted_TestCyl2_A:                  REAL;
  rPressureConverted_TestCyl2_B:                  REAL;
  rPressureConverted_CounterCyl2:                 REAL;
  rPressureConverted_TestCyl3:                    REAL;
  rPressureConverted_TestCyl3_A:                  REAL;
  rPressureConverted_TestCyl3_B:                  REAL;
  rPressureConverted_CounterCyl3:                 REAL;
  rPressureConverted_TestCyl4:                    REAL;
  rPressureConverted_TestCyl4_A:                  REAL;
  rPressureConverted_TestCyl4_B:                  REAL;
  rPressureConverted_CounterCyl4:                 REAL;
{endregion}
  
